// TIA Portal V20 export
FUNCTION_BLOCK "CallEquipment"   // FB44, LAD
TITLE = CallEquipment
// Template of an equipment module. This block contains the logic and futher calls (e.g. sequences, control modules, diagnostics etc.) of the equipment module.
// It can be used out of the box but also adapted to your own needs.
// stored: IsIECCheckEnabled true, MemoryReserve 100, Namespace Unit1.Em5, SetENOAutomatically true
   VAR_INPUT
      ZoneOperationEnable { ExternalWritable := 'False'} : "LWONIK_typeSafetyZoneManualOperation";
      unitEnableControlInterfaces { ExternalWritable := 'False'} : "LAF_typeEnableControlInterfaces";
      commandExcute { ExternalWritable := 'False'} : Bool;
   END_VAR
   VAR_IN_OUT
      unitStatus : "LAF_typeUnitStatus";   // Current unit status o be used in this EM
      emFeedback : "LUC_typeEmFeedback";   // Feedback of the EM to the Unit
      unitAlarmDB : "LAF_typeAlarms";   // Summarized EM Alarms for the Unit
   END_VAR
   VAR
      instSequenceManualInput { ExternalWritable := 'False'} : "Unit1.Em5.Sequence_1_ManualInput";
      instManualInPutInitializedJob1 { ExternalWritable := 'False'} : "LAF_SelectJob";
      instManualInPutLoadingJob2 { ExternalWritable := 'False'} : "LAF_SelectJob";
      instManualInPutUnLoaingJob3 { ExternalWritable := 'False'} : "LAF_SelectJob";
      instCmNgAndManualInputAxisY { ExternalWritable := 'False'} : "LBC_Axis64Pos_TecPlcCn";
      instCmMagazineAxisZ { ExternalWritable := 'False'} : "LBC_Axis64Pos_TecPlcCn";
      instCmNgAndManualInputCylinderUpDown { ExternalWritable := 'False'} : "LBC_TwoWayActuatorCn";
      instcmNgAndManualInputVacuum1OnOff { ExternalWritable := 'False'} : "LBC_TwoWayActuatorCn";
      instCmNgAndManualInputVacuum2OnOff { ExternalWritable := 'False'} : "LBC_TwoWayActuatorCn";
      instCmNgAndManualInputVibrator1OnOff { ExternalWritable := 'False'} : "LBC_TwoWayActuatorCn";
      instCmNgAndManualInputVibrator2OnOff { ExternalWritable := 'False'} : "LBC_TwoWayActuatorCn";
      instcmMagazineLockCylinderUpDown { ExternalWritable := 'False'} : "LBC_TwoWayActuatorCn";
      instCmNgAndManaulInputMagazineElectrodeDetectionSensor { ExternalWritable := 'False'} : "LBC_DigitalSignalCn";
      instCmNgAndManualInputMagazineDetectionSensor { ExternalWritable := 'False'} : "LBC_DigitalSignalCn";
      instCmNgAndManualInputMagazineFullSensor { ExternalWritable := 'False'} : "LBC_DigitalSignalCn";
      instCmNgAndManualInputElectrodeDetectionSensor { ExternalWritable := 'False'} : "LBC_DigitalSignalCn";
      instcmMagazineSafetyPinIdlePosition { ExternalWritable := 'False'} : "LBC_DigitalSignalCn";
      instNgAndManualInputAxisControlInterlockSummary { ExternalWritable := 'False'} : "LER_Axis64Pos_InterlockSummary";
      instMagazineAxisControlInterlockSummary { ExternalWritable := 'False'} : "LER_Axis64Pos_InterlockSummary";
      instServoTorqueCal_DR7 { ExternalWritable := 'False'} : "LER_ServoTorqueCal";
      instServoTorqueCal_DR8 { ExternalWritable := 'False'} : "LER_ServoTorqueCal";
      instLDrv701ControlMagazineAxisZ { ExternalWritable := 'False'} : "LDrvSafe_SinaTlg701Control";   // Drive Telegram Function Library
      instLDrv701StatusMagazineAxisZ { ExternalWritable := 'False'} : "LDrvSafe_SinaTlg701Status";   // Drive Telegram Function Library
      statUnitStatus { ExternalWritable := 'False'} : "LAF_typeUnitStatus";   // Unit Status used in this EM
      statAllBrakeTest { ExternalWritable := 'False'} : "LER_typeBrakeTestUnitCommands";
      instManageAlarms { ExternalWritable := 'False'} : "LAF_ManageAlarms";
      instEventsPFE { S7_SetPoint := 'True'} : "Unit1.Em5.EventsPFE";
      statPulse { ExternalWritable := 'False'} : Array[0..99] of Bool;
      statTonTimer { ExternalWritable := 'False'} : Array[0..99] of TON_TIME;
      statTofTimer { ExternalWritable := 'False'} : Array[0..99] of TOF_TIME;
      statEnableManualCmds { ExternalWritable := 'False'} : Bool;
      LoadingCount { ExternalWritable := 'False'} : Int;
   END_VAR
   VAR_TEMP
      tempScInProduction : Bool;   // Mode Production and StateComplete
      tempScNoProduction : Bool;   // Mode Manual and StateComplete
   END_VAR
   VAR CONSTANT
      TO_DO_INSERT_PRECONDITIONS_HERE : Bool := TRUE;   // Template : Add em specific conditions here
      NO_JOB : DInt;   // No job
      TRUE : Bool := TRUE;
      FALSE : Bool := FALSE;
      INIT_POSITION_NUMBER : SInt := -1;
      MIN_POSITION_NUMBER : SInt;
   END_VAR
   VAR_TEMP   // added for the SCL form of the ladder/FBD networks
      _w1 : Bool;
      _w2 : Bool;
      _w3 : Bool;
      _w4 : Bool;
      _w5 : Bool;
      _w6 : Bool;
      _w7 : Bool;
      _w8 : Bool;
      _w9 : Bool;
      _w10 : Bool;
      _w11 : Bool;
      _w12 : Bool;
      _w13 : Bool;
      _w14 : Bool;
      _w15 : Bool;
      _w16 : Bool;
   END_VAR
BEGIN

REGION Network 1: BLOCK INFO HEADER
   // (company) / (C) Copyright (year)
   // ---------------------------------------------------------------------------------
   // Title:                             (Title of this block)
   // Comment/Function: (that is implemented in the block)
   // Library/Family:           (that the source is dedicated to)
   // Author:                        (department / person in charge / contact)
   // Target System:          (test system with FW version)
   // Engineering:              TIA Portal (SW version)
   // Restrictions:               (OB types, etc.)
   // Requirements:           (hardware, technological package, etc.)
   // ---------------------------------------------------------------------------------
   // Change log table:
   // Version          | Date             | Signature      | Expert in charge  | Changes applied ------------------------|----------------------|-------------------------|--------------------------------|-----------------------
   // 001.000.000 | yyyy-mm-dd | 0x00000000 | (name of expert) | First released version
END_REGION

REGION Network 2: DESCRIPTION
   // This is a template block provided by the Automation Framework. It can be used to create an own project.
   // The Block Info Header is prepared to put in your own data.
   // Description of the block could be added here and the docu created by Code2Docu.
END_REGION

REGION Network 3: ******************** Unit Input ********************
END_REGION

REGION Network 4: Em Nodes Brake Test
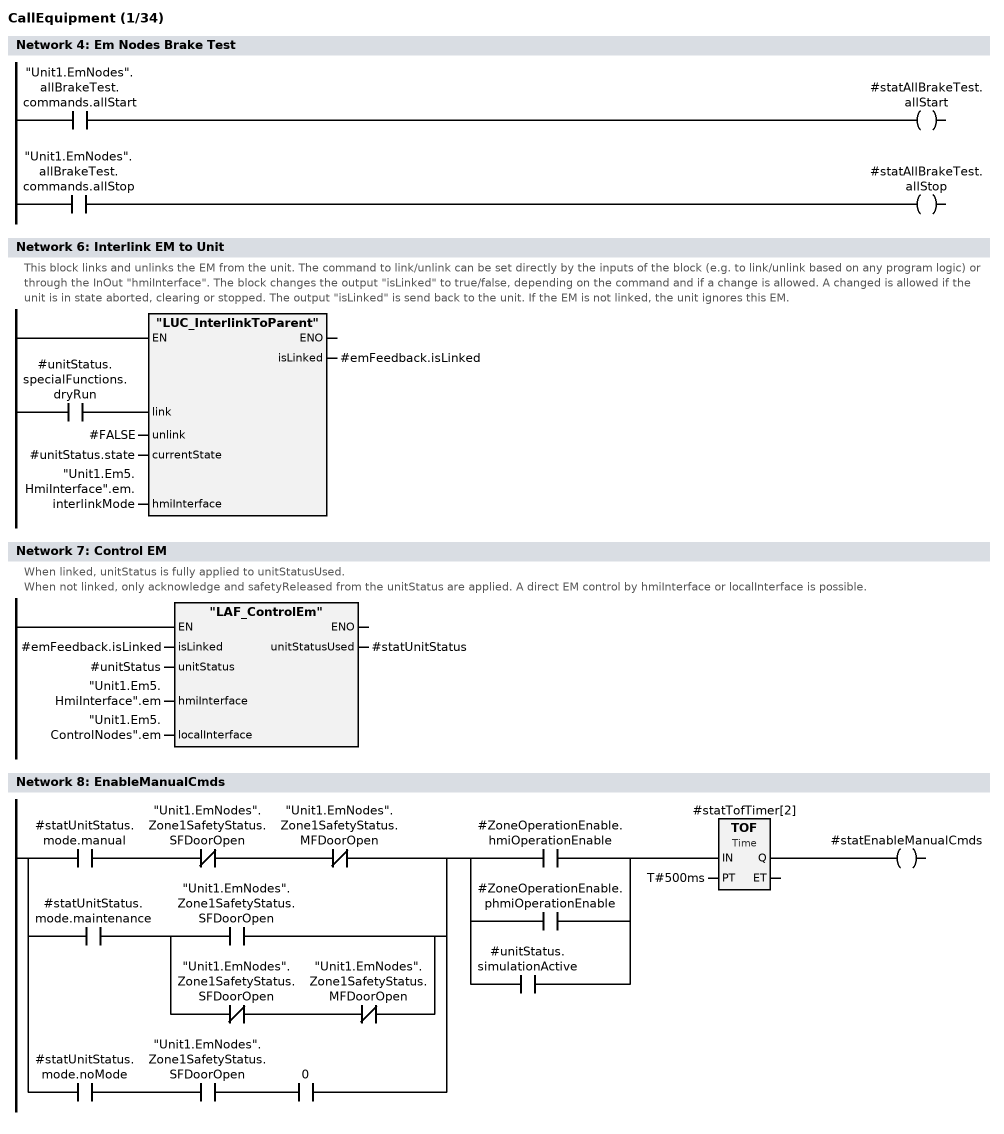
   RUNG wire#powerrail
      Contact( "Unit1.EmNodes".allBrakeTest.commands.allStart )
      Coil( #statAllBrakeTest.allStart )
   END_RUNG
   RUNG wire#powerrail
      Contact( "Unit1.EmNodes".allBrakeTest.commands.allStop )
      Coil( #statAllBrakeTest.allStop )
   END_RUNG
   // the same network as SCL:
   #statAllBrakeTest.allStart := "Unit1.EmNodes".allBrakeTest.commands.allStart;
   #statAllBrakeTest.allStop := "Unit1.EmNodes".allBrakeTest.commands.allStop;
END_REGION

REGION Network 5: ******************** Equipment Control ********************
END_REGION

REGION Network 6: Interlink EM to Unit
   // This block links and unlinks the EM from the unit. The command to link/unlink can be set directly by the inputs of the block (e.g. to link/unlink based on any program logic) or through the InOut "hmiInterface". The block changes the output "isLinked" to true/false, depending on the command and if a change is allowed. A changed is allowed if the unit is in state aborted, clearing or stopped. The output "isLinked" is send back to the unit. If the EM is not linked, the unit ignores this EM.
   RUNG wire#powerrail
      "LUC_InterlinkToParent"(link := wire#w1, unlink := #FALSE, currentState := #unitStatus.state, hmiInterface := "Unit1.Em5.HmiInterface".em.interlinkMode, isLinked => #emFeedback.isLinked)
   END_RUNG
   RUNG wire#powerrail
      Contact( #unitStatus.specialFunctions.dryRun )
   END_RUNG wire#w1
   // the same network as SCL:
   "LUC_InterlinkToParent"(link := #unitStatus.specialFunctions.dryRun,
                           unlink := #FALSE,
                           currentState := #unitStatus.state,
                           hmiInterface := "Unit1.Em5.HmiInterface".em.interlinkMode,
                           isLinked => #emFeedback.isLinked);
END_REGION

REGION Network 7: Control EM
   // When linked, unitStatus is fully applied to unitStatusUsed.
   // When not linked, only acknowledge and safetyReleased from the unitStatus are applied. A direct EM control by hmiInterface or localInterface is possible.
   RUNG wire#powerrail
      "LAF_ControlEm"(isLinked := #emFeedback.isLinked, unitStatus := #unitStatus, hmiInterface := "Unit1.Em5.HmiInterface".em, localInterface := "Unit1.Em5.ControlNodes".em, unitStatusUsed => #statUnitStatus)
   END_RUNG
   // the same network as SCL:
   "LAF_ControlEm"(isLinked := #emFeedback.isLinked,
                   unitStatus := #unitStatus,
                   hmiInterface := "Unit1.Em5.HmiInterface".em,
                   localInterface := "Unit1.Em5.ControlNodes".em,
                   unitStatusUsed => #statUnitStatus);
END_REGION

REGION Network 8: EnableManualCmds
   RUNG wire#powerrail
      Contact( #statUnitStatus.mode.manual )
      I_Contact( "Unit1.EmNodes".Zone1SafetyStatus.SFDoorOpen )
      I_Contact( "Unit1.EmNodes".Zone1SafetyStatus.MFDoorOpen )
      wire#w1
      Contact( #ZoneOperationEnable.hmiOperationEnable )
      wire#w3
      { S7_Templates := "time_type := Time" } #statTofTimer[2].TOF(pt := T#500ms, et =>)
      Coil( #statEnableManualCmds )
   END_RUNG
   RUNG wire#powerrail
      Contact( #statUnitStatus.mode.maintenance )
      wire#w2
      Contact( "Unit1.EmNodes".Zone1SafetyStatus.SFDoorOpen )
   END_RUNG wire#w1
   RUNG wire#w2
      I_Contact( "Unit1.EmNodes".Zone1SafetyStatus.SFDoorOpen )
      I_Contact( "Unit1.EmNodes".Zone1SafetyStatus.MFDoorOpen )
   END_RUNG wire#w1
   RUNG wire#powerrail
      Contact( #statUnitStatus.mode.noMode )
      Contact( "Unit1.EmNodes".Zone1SafetyStatus.SFDoorOpen )
      Contact( 0 )
   END_RUNG wire#w1
   RUNG wire#w1
      Contact( #ZoneOperationEnable.phmiOperationEnable )
   END_RUNG wire#w3
   RUNG wire#w1
      Contact( #unitStatus.simulationActive )
   END_RUNG wire#w3
   // the same network as SCL:
   #statTofTimer[2].TOF(IN := ((#statUnitStatus.mode.manual AND NOT "Unit1.EmNodes".Zone1SafetyStatus.SFDoorOpen AND NOT "Unit1.EmNodes".Zone1SafetyStatus.MFDoorOpen) OR (#statUnitStatus.mode.maintenance AND ("Unit1.EmNodes".Zone1SafetyStatus.SFDoorOpen OR (NOT "Unit1.EmNodes".Zone1SafetyStatus.SFDoorOpen AND NOT "Unit1.EmNodes".Zone1SafetyStatus.MFDoorOpen))) OR (#statUnitStatus.mode.noMode AND "Unit1.EmNodes".Zone1SafetyStatus.SFDoorOpen AND 0)) AND (#ZoneOperationEnable.hmiOperationEnable OR #ZoneOperationEnable.phmiOperationEnable OR #unitStatus.simulationActive),
                        PT := T#500ms);
   #statEnableManualCmds := #statTofTimer[2].Q;
END_REGION

REGION Network 9: Alarms Disabled
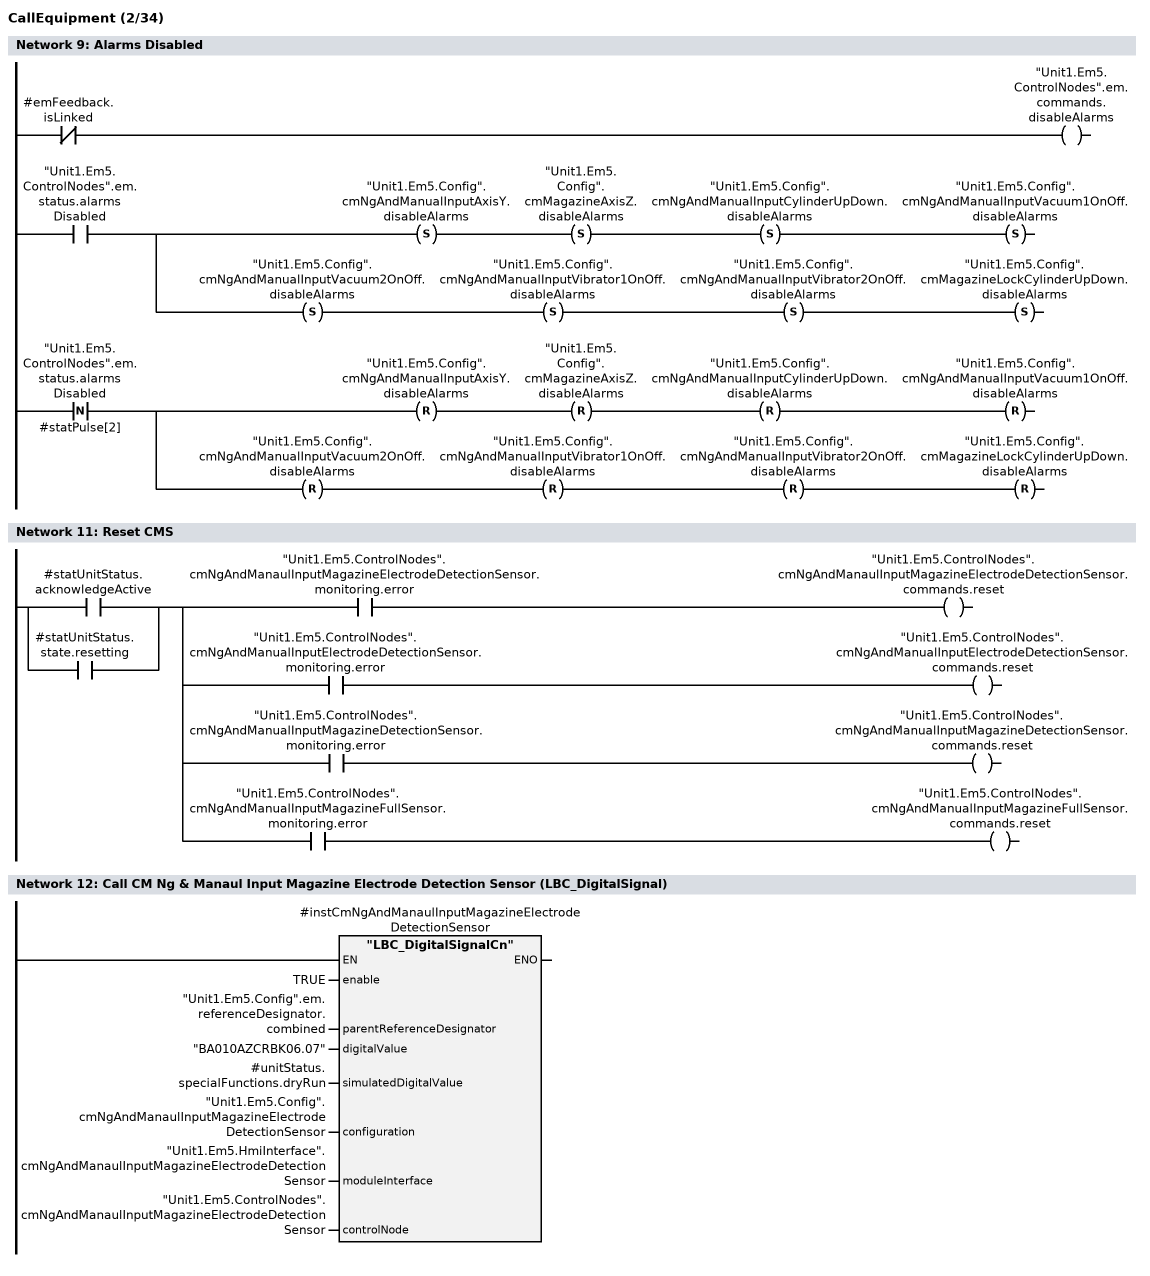
   RUNG wire#powerrail
      I_Contact( #emFeedback.isLinked )
      Coil( "Unit1.Em5.ControlNodes".em.commands.disableAlarms )
   END_RUNG
   RUNG wire#powerrail
      Contact( "Unit1.Em5.ControlNodes".em.status.alarmsDisabled )
      wire#w1
      S_Coil( "Unit1.Em5.Config".cmNgAndManualInputAxisY.disableAlarms )
      S_Coil( "Unit1.Em5.Config".cmMagazineAxisZ.disableAlarms )
      S_Coil( "Unit1.Em5.Config".cmNgAndManualInputCylinderUpDown.disableAlarms )
      S_Coil( "Unit1.Em5.Config".cmNgAndManualInputVacuum1OnOff.disableAlarms )
   END_RUNG
   RUNG wire#w1
      S_Coil( "Unit1.Em5.Config".cmNgAndManualInputVacuum2OnOff.disableAlarms )
      S_Coil( "Unit1.Em5.Config".cmNgAndManualInputVibrator1OnOff.disableAlarms )
      S_Coil( "Unit1.Em5.Config".cmNgAndManualInputVibrator2OnOff.disableAlarms )
      S_Coil( "Unit1.Em5.Config".cmMagazineLockCylinderUpDown.disableAlarms )
   END_RUNG
   RUNG wire#powerrail
      N_Contact(operand := "Unit1.Em5.ControlNodes".em.status.alarmsDisabled, bit := #statPulse[2])
      wire#w2
      R_Coil( "Unit1.Em5.Config".cmNgAndManualInputAxisY.disableAlarms )
      R_Coil( "Unit1.Em5.Config".cmMagazineAxisZ.disableAlarms )
      R_Coil( "Unit1.Em5.Config".cmNgAndManualInputCylinderUpDown.disableAlarms )
      R_Coil( "Unit1.Em5.Config".cmNgAndManualInputVacuum1OnOff.disableAlarms )
   END_RUNG
   RUNG wire#w2
      R_Coil( "Unit1.Em5.Config".cmNgAndManualInputVacuum2OnOff.disableAlarms )
      R_Coil( "Unit1.Em5.Config".cmNgAndManualInputVibrator1OnOff.disableAlarms )
      R_Coil( "Unit1.Em5.Config".cmNgAndManualInputVibrator2OnOff.disableAlarms )
      R_Coil( "Unit1.Em5.Config".cmMagazineLockCylinderUpDown.disableAlarms )
   END_RUNG
   // the same network as SCL:
   "Unit1.Em5.ControlNodes".em.commands.disableAlarms := NOT #emFeedback.isLinked;
   IF "Unit1.Em5.ControlNodes".em.status.alarmsDisabled THEN
       "Unit1.Em5.Config".cmNgAndManualInputAxisY.disableAlarms := TRUE;
       "Unit1.Em5.Config".cmMagazineAxisZ.disableAlarms := TRUE;
       "Unit1.Em5.Config".cmNgAndManualInputCylinderUpDown.disableAlarms := TRUE;
       "Unit1.Em5.Config".cmNgAndManualInputVacuum1OnOff.disableAlarms := TRUE;
       "Unit1.Em5.Config".cmNgAndManualInputVacuum2OnOff.disableAlarms := TRUE;
       "Unit1.Em5.Config".cmNgAndManualInputVibrator1OnOff.disableAlarms := TRUE;
       "Unit1.Em5.Config".cmNgAndManualInputVibrator2OnOff.disableAlarms := TRUE;
       "Unit1.Em5.Config".cmMagazineLockCylinderUpDown.disableAlarms := TRUE;
   END_IF;
   #_w1 := NOT "Unit1.Em5.ControlNodes".em.status.alarmsDisabled AND #statPulse[2];   // falling edge of "Unit1.Em5.ControlNodes".em.status.alarmsDisabled
   #statPulse[2] := "Unit1.Em5.ControlNodes".em.status.alarmsDisabled;
   IF #_w1 THEN
       "Unit1.Em5.Config".cmNgAndManualInputAxisY.disableAlarms := FALSE;
       "Unit1.Em5.Config".cmMagazineAxisZ.disableAlarms := FALSE;
       "Unit1.Em5.Config".cmNgAndManualInputCylinderUpDown.disableAlarms := FALSE;
       "Unit1.Em5.Config".cmNgAndManualInputVacuum1OnOff.disableAlarms := FALSE;
       "Unit1.Em5.Config".cmNgAndManualInputVacuum2OnOff.disableAlarms := FALSE;
       "Unit1.Em5.Config".cmNgAndManualInputVibrator1OnOff.disableAlarms := FALSE;
       "Unit1.Em5.Config".cmNgAndManualInputVibrator2OnOff.disableAlarms := FALSE;
       "Unit1.Em5.Config".cmMagazineLockCylinderUpDown.disableAlarms := FALSE;
   END_IF;
END_REGION

REGION Network 10: ******************** Control Modules (Sensors) ********************
   // Call control modules that are sensors before the em logic (jobs and sequence), so that the latest value is used in the logic.
END_REGION

REGION Network 11: Reset CMS
   RUNG wire#powerrail
      Contact( #statUnitStatus.acknowledgeActive )
      wire#w1
      Contact( "Unit1.Em5.ControlNodes".cmNgAndManaulInputMagazineElectrodeDetectionSensor.monitoring.error )
      Coil( "Unit1.Em5.ControlNodes".cmNgAndManaulInputMagazineElectrodeDetectionSensor.commands.reset )
   END_RUNG
   RUNG wire#powerrail
      Contact( #statUnitStatus.state.resetting )
   END_RUNG wire#w1
   RUNG wire#w1
      Contact( "Unit1.Em5.ControlNodes".cmNgAndManualInputElectrodeDetectionSensor.monitoring.error )
      Coil( "Unit1.Em5.ControlNodes".cmNgAndManualInputElectrodeDetectionSensor.commands.reset )
   END_RUNG
   RUNG wire#w1
      Contact( "Unit1.Em5.ControlNodes".cmNgAndManualInputMagazineDetectionSensor.monitoring.error )
      Coil( "Unit1.Em5.ControlNodes".cmNgAndManualInputMagazineDetectionSensor.commands.reset )
   END_RUNG
   RUNG wire#w1
      Contact( "Unit1.Em5.ControlNodes".cmNgAndManualInputMagazineFullSensor.monitoring.error )
      Coil( "Unit1.Em5.ControlNodes".cmNgAndManualInputMagazineFullSensor.commands.reset )
   END_RUNG
   // the same network as SCL:
   #_w1 := #statUnitStatus.acknowledgeActive OR #statUnitStatus.state.resetting;
   "Unit1.Em5.ControlNodes".cmNgAndManaulInputMagazineElectrodeDetectionSensor.commands.reset := #_w1 AND "Unit1.Em5.ControlNodes".cmNgAndManaulInputMagazineElectrodeDetectionSensor.monitoring.error;
   "Unit1.Em5.ControlNodes".cmNgAndManualInputElectrodeDetectionSensor.commands.reset := #_w1 AND "Unit1.Em5.ControlNodes".cmNgAndManualInputElectrodeDetectionSensor.monitoring.error;
   "Unit1.Em5.ControlNodes".cmNgAndManualInputMagazineDetectionSensor.commands.reset := #_w1 AND "Unit1.Em5.ControlNodes".cmNgAndManualInputMagazineDetectionSensor.monitoring.error;
   "Unit1.Em5.ControlNodes".cmNgAndManualInputMagazineFullSensor.commands.reset := #_w1 AND "Unit1.Em5.ControlNodes".cmNgAndManualInputMagazineFullSensor.monitoring.error;
END_REGION

REGION Network 12: Call CM Ng & Manaul Input Magazine Electrode Detection Sensor (LBC_DigitalSignal)
   RUNG wire#powerrail
      #instCmNgAndManaulInputMagazineElectrodeDetectionSensor(enable := TRUE, parentReferenceDesignator := "Unit1.Em5.Config".em.referenceDesignator.combined, digitalValue := "BA010AZCRBK06.07", simulatedDigitalValue := #unitStatus.specialFunctions.dryRun, configuration := "Unit1.Em5.Config".cmNgAndManaulInputMagazineElectrodeDetectionSensor, moduleInterface := "Unit1.Em5.HmiInterface".cmNgAndManaulInputMagazineElectrodeDetectionSensor, controlNode := "Unit1.Em5.ControlNodes".cmNgAndManaulInputMagazineElectrodeDetectionSensor)
   END_RUNG
   // the same network as SCL:
   #instCmNgAndManaulInputMagazineElectrodeDetectionSensor(enable := TRUE,   // "LBC_DigitalSignalCn"
                           parentReferenceDesignator := "Unit1.Em5.Config".em.referenceDesignator.combined,
                           digitalValue := "BA010AZCRBK06.07",
                           simulatedDigitalValue := #unitStatus.specialFunctions.dryRun,
                           configuration := "Unit1.Em5.Config".cmNgAndManaulInputMagazineElectrodeDetectionSensor,
                           moduleInterface := "Unit1.Em5.HmiInterface".cmNgAndManaulInputMagazineElectrodeDetectionSensor,
                           controlNode := "Unit1.Em5.ControlNodes".cmNgAndManaulInputMagazineElectrodeDetectionSensor);
END_REGION

REGION Network 13: Call CM Ng & Manaul Input Magazine Detection Sensor (LBC_DigitalSignal)
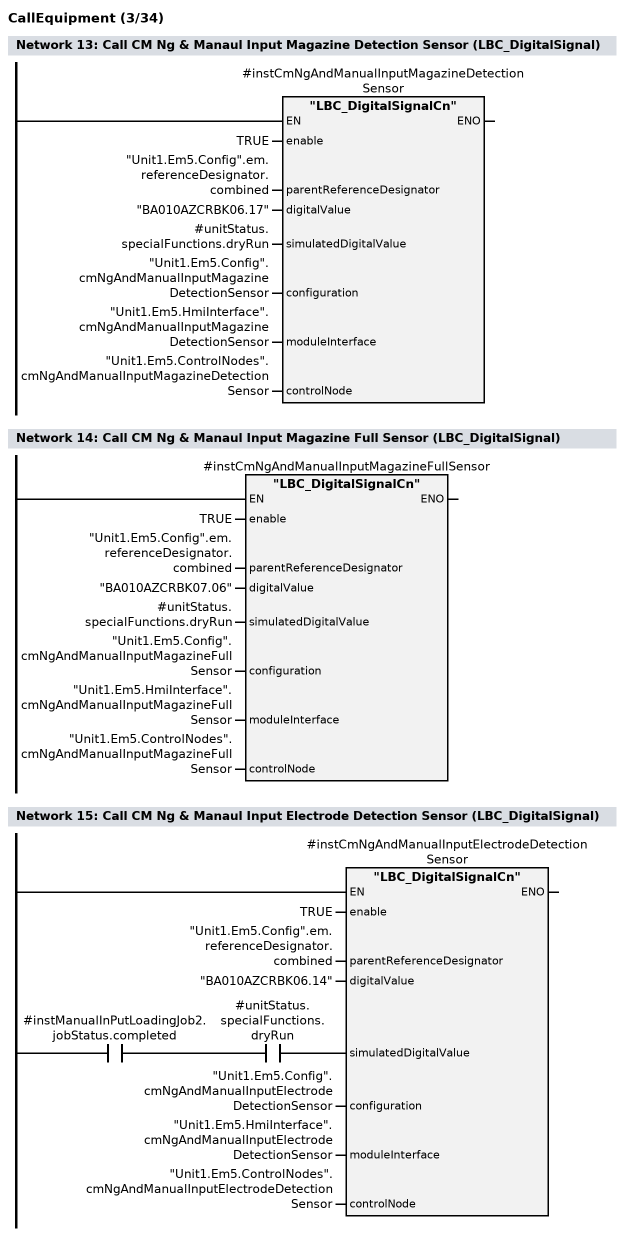
   RUNG wire#powerrail
      #instCmNgAndManualInputMagazineDetectionSensor(enable := TRUE, parentReferenceDesignator := "Unit1.Em5.Config".em.referenceDesignator.combined, digitalValue := "BA010AZCRBK06.17", simulatedDigitalValue := #unitStatus.specialFunctions.dryRun, configuration := "Unit1.Em5.Config".cmNgAndManualInputMagazineDetectionSensor, moduleInterface := "Unit1.Em5.HmiInterface".cmNgAndManualInputMagazineDetectionSensor, controlNode := "Unit1.Em5.ControlNodes".cmNgAndManualInputMagazineDetectionSensor)
   END_RUNG
   // the same network as SCL:
   #instCmNgAndManualInputMagazineDetectionSensor(enable := TRUE,   // "LBC_DigitalSignalCn"
                           parentReferenceDesignator := "Unit1.Em5.Config".em.referenceDesignator.combined,
                           digitalValue := "BA010AZCRBK06.17",
                           simulatedDigitalValue := #unitStatus.specialFunctions.dryRun,
                           configuration := "Unit1.Em5.Config".cmNgAndManualInputMagazineDetectionSensor,
                           moduleInterface := "Unit1.Em5.HmiInterface".cmNgAndManualInputMagazineDetectionSensor,
                           controlNode := "Unit1.Em5.ControlNodes".cmNgAndManualInputMagazineDetectionSensor);
END_REGION

REGION Network 14: Call CM Ng & Manaul Input Magazine Full Sensor (LBC_DigitalSignal)
   RUNG wire#powerrail
      #instCmNgAndManualInputMagazineFullSensor(enable := TRUE, parentReferenceDesignator := "Unit1.Em5.Config".em.referenceDesignator.combined, digitalValue := "BA010AZCRBK07.06", simulatedDigitalValue := #unitStatus.specialFunctions.dryRun, configuration := "Unit1.Em5.Config".cmNgAndManualInputMagazineFullSensor, moduleInterface := "Unit1.Em5.HmiInterface".cmNgAndManualInputMagazineFullSensor, controlNode := "Unit1.Em5.ControlNodes".cmNgAndManualInputMagazineFullSensor)
   END_RUNG
   // the same network as SCL:
   #instCmNgAndManualInputMagazineFullSensor(enable := TRUE,   // "LBC_DigitalSignalCn"
                           parentReferenceDesignator := "Unit1.Em5.Config".em.referenceDesignator.combined,
                           digitalValue := "BA010AZCRBK07.06",
                           simulatedDigitalValue := #unitStatus.specialFunctions.dryRun,
                           configuration := "Unit1.Em5.Config".cmNgAndManualInputMagazineFullSensor,
                           moduleInterface := "Unit1.Em5.HmiInterface".cmNgAndManualInputMagazineFullSensor,
                           controlNode := "Unit1.Em5.ControlNodes".cmNgAndManualInputMagazineFullSensor);
END_REGION

REGION Network 15: Call CM Ng & Manaul Input Electrode Detection Sensor (LBC_DigitalSignal)
   RUNG wire#powerrail
      #instCmNgAndManualInputElectrodeDetectionSensor(simulatedDigitalValue := wire#w1, enable := TRUE, parentReferenceDesignator := "Unit1.Em5.Config".em.referenceDesignator.combined, digitalValue := "BA010AZCRBK06.14", configuration := "Unit1.Em5.Config".cmNgAndManualInputElectrodeDetectionSensor, moduleInterface := "Unit1.Em5.HmiInterface".cmNgAndManualInputElectrodeDetectionSensor, controlNode := "Unit1.Em5.ControlNodes".cmNgAndManualInputElectrodeDetectionSensor)
   END_RUNG
   RUNG wire#powerrail
      Contact( #instManualInPutLoadingJob2.jobStatus.completed )
      Contact( #unitStatus.specialFunctions.dryRun )
   END_RUNG wire#w1
   // the same network as SCL:
   #instCmNgAndManualInputElectrodeDetectionSensor(enable := TRUE,   // "LBC_DigitalSignalCn"
                           parentReferenceDesignator := "Unit1.Em5.Config".em.referenceDesignator.combined,
                           digitalValue := "BA010AZCRBK06.14",
                           simulatedDigitalValue := #instManualInPutLoadingJob2.jobStatus.completed AND #unitStatus.specialFunctions.dryRun,
                           configuration := "Unit1.Em5.Config".cmNgAndManualInputElectrodeDetectionSensor,
                           moduleInterface := "Unit1.Em5.HmiInterface".cmNgAndManualInputElectrodeDetectionSensor,
                           controlNode := "Unit1.Em5.ControlNodes".cmNgAndManualInputElectrodeDetectionSensor);
END_REGION

REGION Network 16: Call CM Magazine Safety Pin Idle Position (LBC_DigitalSignal)
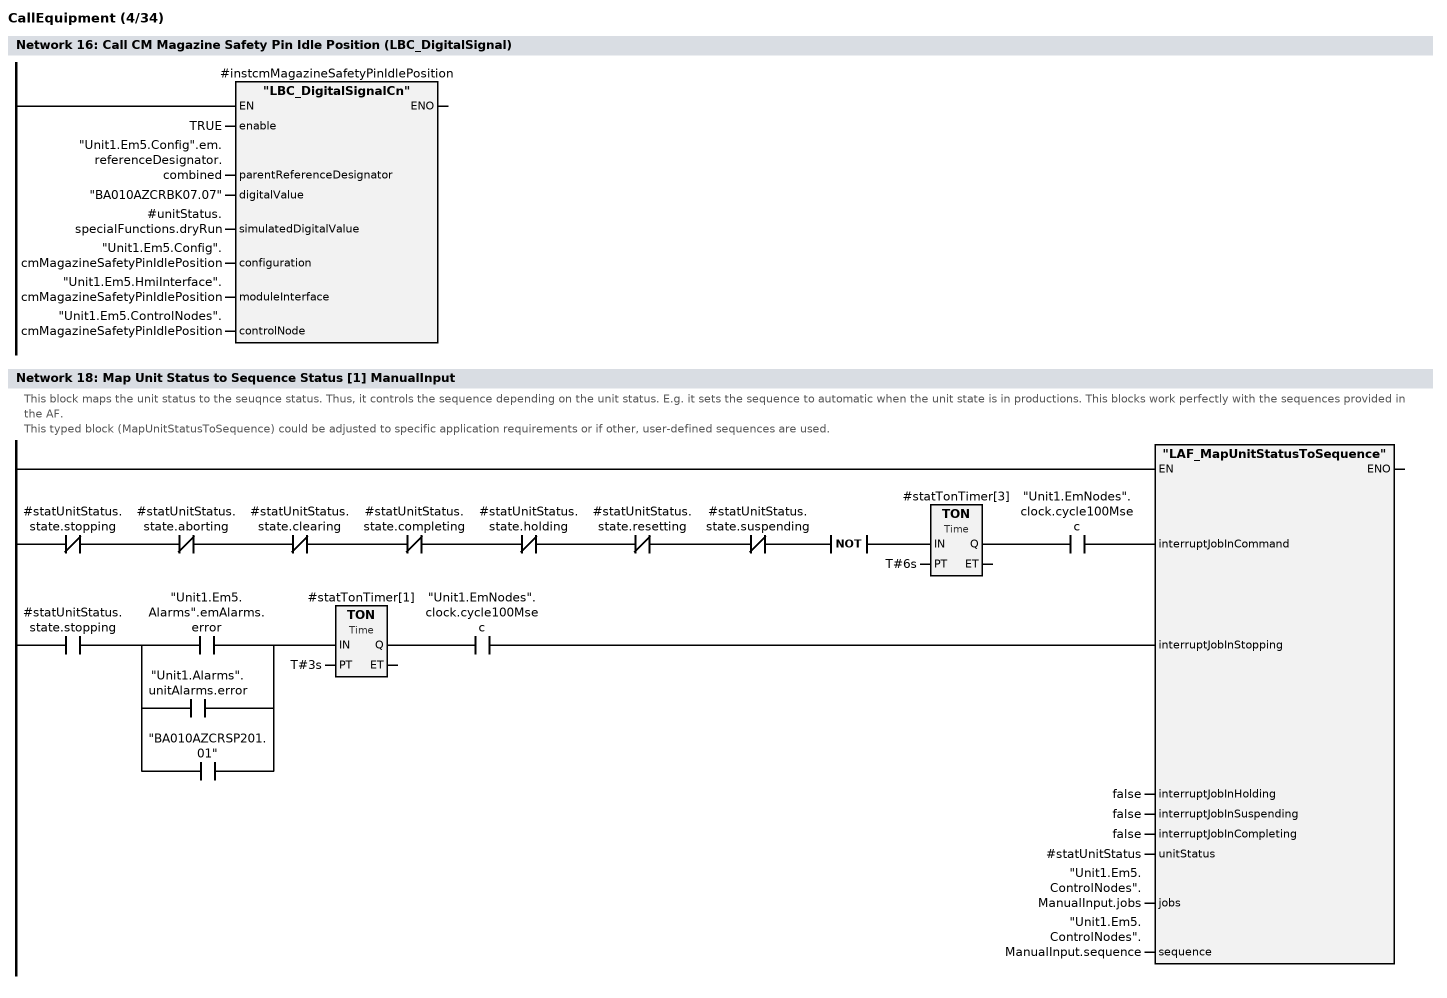
   RUNG wire#powerrail
      #instcmMagazineSafetyPinIdlePosition(enable := TRUE, parentReferenceDesignator := "Unit1.Em5.Config".em.referenceDesignator.combined, digitalValue := "BA010AZCRBK07.07", simulatedDigitalValue := #unitStatus.specialFunctions.dryRun, configuration := "Unit1.Em5.Config".cmMagazineSafetyPinIdlePosition, moduleInterface := "Unit1.Em5.HmiInterface".cmMagazineSafetyPinIdlePosition, controlNode := "Unit1.Em5.ControlNodes".cmMagazineSafetyPinIdlePosition)
   END_RUNG
   // the same network as SCL:
   #instcmMagazineSafetyPinIdlePosition(enable := TRUE,   // "LBC_DigitalSignalCn"
                           parentReferenceDesignator := "Unit1.Em5.Config".em.referenceDesignator.combined,
                           digitalValue := "BA010AZCRBK07.07",
                           simulatedDigitalValue := #unitStatus.specialFunctions.dryRun,
                           configuration := "Unit1.Em5.Config".cmMagazineSafetyPinIdlePosition,
                           moduleInterface := "Unit1.Em5.HmiInterface".cmMagazineSafetyPinIdlePosition,
                           controlNode := "Unit1.Em5.ControlNodes".cmMagazineSafetyPinIdlePosition);
END_REGION

REGION Network 17: ******************** Equipment Logic ********************
END_REGION

REGION Network 18: Map Unit Status to Sequence Status [1] ManualInput
   // This block maps the unit status to the seuqnce status. Thus, it controls the sequence depending on the unit status. E.g. it sets the sequence to automatic when the unit state is in productions. This blocks work perfectly with the sequences provided in the AF. 
   // This typed block (MapUnitStatusToSequence) could be adjusted to specific application requirements or if other, user-defined sequences are used.
   RUNG wire#powerrail
      "LAF_MapUnitStatusToSequence"(interruptJobInCommand := wire#w1, interruptJobInStopping := wire#w4, interruptJobInHolding := false, interruptJobInSuspending := false, interruptJobInCompleting := false, unitStatus := #statUnitStatus, jobs := "Unit1.Em5.ControlNodes".ManualInput.jobs, sequence := "Unit1.Em5.ControlNodes".ManualInput.sequence)
   END_RUNG
   RUNG wire#powerrail
      I_Contact( #statUnitStatus.state.stopping )
      I_Contact( #statUnitStatus.state.aborting )
      I_Contact( #statUnitStatus.state.clearing )
      I_Contact( #statUnitStatus.state.completing )
      I_Contact( #statUnitStatus.state.holding )
      I_Contact( #statUnitStatus.state.resetting )
      I_Contact( #statUnitStatus.state.suspending )
      Not()
      { S7_Templates := "time_type := Time" } #statTonTimer[3].TON(pt := T#6s, et =>)
      Contact( "Unit1.EmNodes".clock.cycle100Msec )
   END_RUNG wire#w1
   RUNG wire#powerrail
      Contact( #statUnitStatus.state.stopping )
      wire#w2
      Contact( "Unit1.Em5.Alarms".emAlarms.error )
      wire#w3
      { S7_Templates := "time_type := Time" } #statTonTimer[1].TON(pt := T#3s, et =>)
      Contact( "Unit1.EmNodes".clock.cycle100Msec )
   END_RUNG wire#w4
   RUNG wire#w2
      Contact( "Unit1.Alarms".unitAlarms.error )
   END_RUNG wire#w3
   RUNG wire#w2
      Contact( "BA010AZCRSP201.01" )
   END_RUNG wire#w3
   // the same network as SCL:
   #statTonTimer[3].TON(IN := NOT (NOT #statUnitStatus.state.stopping AND NOT #statUnitStatus.state.aborting AND NOT #statUnitStatus.state.clearing AND NOT #statUnitStatus.state.completing AND NOT #statUnitStatus.state.holding AND NOT #statUnitStatus.state.resetting AND NOT #statUnitStatus.state.suspending),
                        PT := T#6s);
   #_w1 := #statTonTimer[3].Q AND "Unit1.EmNodes".clock.cycle100Msec;
   #statTonTimer[1].TON(IN := #statUnitStatus.state.stopping AND ("Unit1.Em5.Alarms".emAlarms.error OR "Unit1.Alarms".unitAlarms.error OR "BA010AZCRSP201.01"),
                        PT := T#3s);
   "LAF_MapUnitStatusToSequence"(interruptJobInCommand := #_w1,
                           interruptJobInStopping := #statTonTimer[1].Q AND "Unit1.EmNodes".clock.cycle100Msec,
                           interruptJobInHolding := false,
                           interruptJobInSuspending := false,
                           interruptJobInCompleting := false,
                           unitStatus := #statUnitStatus,
                           jobs := "Unit1.Em5.ControlNodes".ManualInput.jobs,
                           sequence := "Unit1.Em5.ControlNodes".ManualInput.sequence);
END_REGION

REGION Network 19: Select Job [1] ManualInput Initialized
   // Decide which Step Sequence to start depending on the OMAC State and EM conditions
   // First Move Block is to Initialize the jobSelect Number
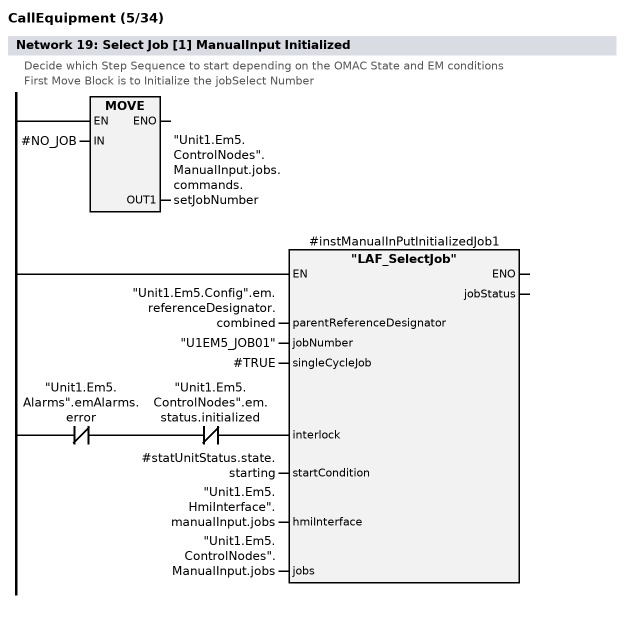
   RUNG wire#powerrail
      Move(in := #NO_JOB, out1 => "Unit1.Em5.ControlNodes".ManualInput.jobs.commands.setJobNumber)
   END_RUNG
   RUNG wire#powerrail
      #instManualInPutInitializedJob1(interlock := wire#w1, parentReferenceDesignator := "Unit1.Em5.Config".em.referenceDesignator.combined, jobNumber := "U1EM5_JOB01", singleCycleJob := #TRUE, startCondition := #statUnitStatus.state.starting, hmiInterface := "Unit1.Em5.HmiInterface".manualInput.jobs, jobs := "Unit1.Em5.ControlNodes".ManualInput.jobs, jobStatus =>)
   END_RUNG
   RUNG wire#powerrail
      I_Contact( "Unit1.Em5.Alarms".emAlarms.error )
      I_Contact( "Unit1.Em5.ControlNodes".em.status.initialized )
   END_RUNG wire#w1
   // the same network as SCL:
   "Unit1.Em5.ControlNodes".ManualInput.jobs.commands.setJobNumber := #NO_JOB;
   #instManualInPutInitializedJob1(parentReferenceDesignator := "Unit1.Em5.Config".em.referenceDesignator.combined,   // "LAF_SelectJob"
                           jobNumber := "U1EM5_JOB01",
                           singleCycleJob := #TRUE,
                           interlock := NOT "Unit1.Em5.Alarms".emAlarms.error AND NOT "Unit1.Em5.ControlNodes".em.status.initialized,
                           startCondition := #statUnitStatus.state.starting,
                           hmiInterface := "Unit1.Em5.HmiInterface".manualInput.jobs,
                           jobs := "Unit1.Em5.ControlNodes".ManualInput.jobs);
END_REGION

REGION Network 20: Select Job [2] Loading Auto
   // Decide which Step Sequence to start depending on the OMAC State and EM conditions
   // First Move Block is to Initialize the jobSelect Number
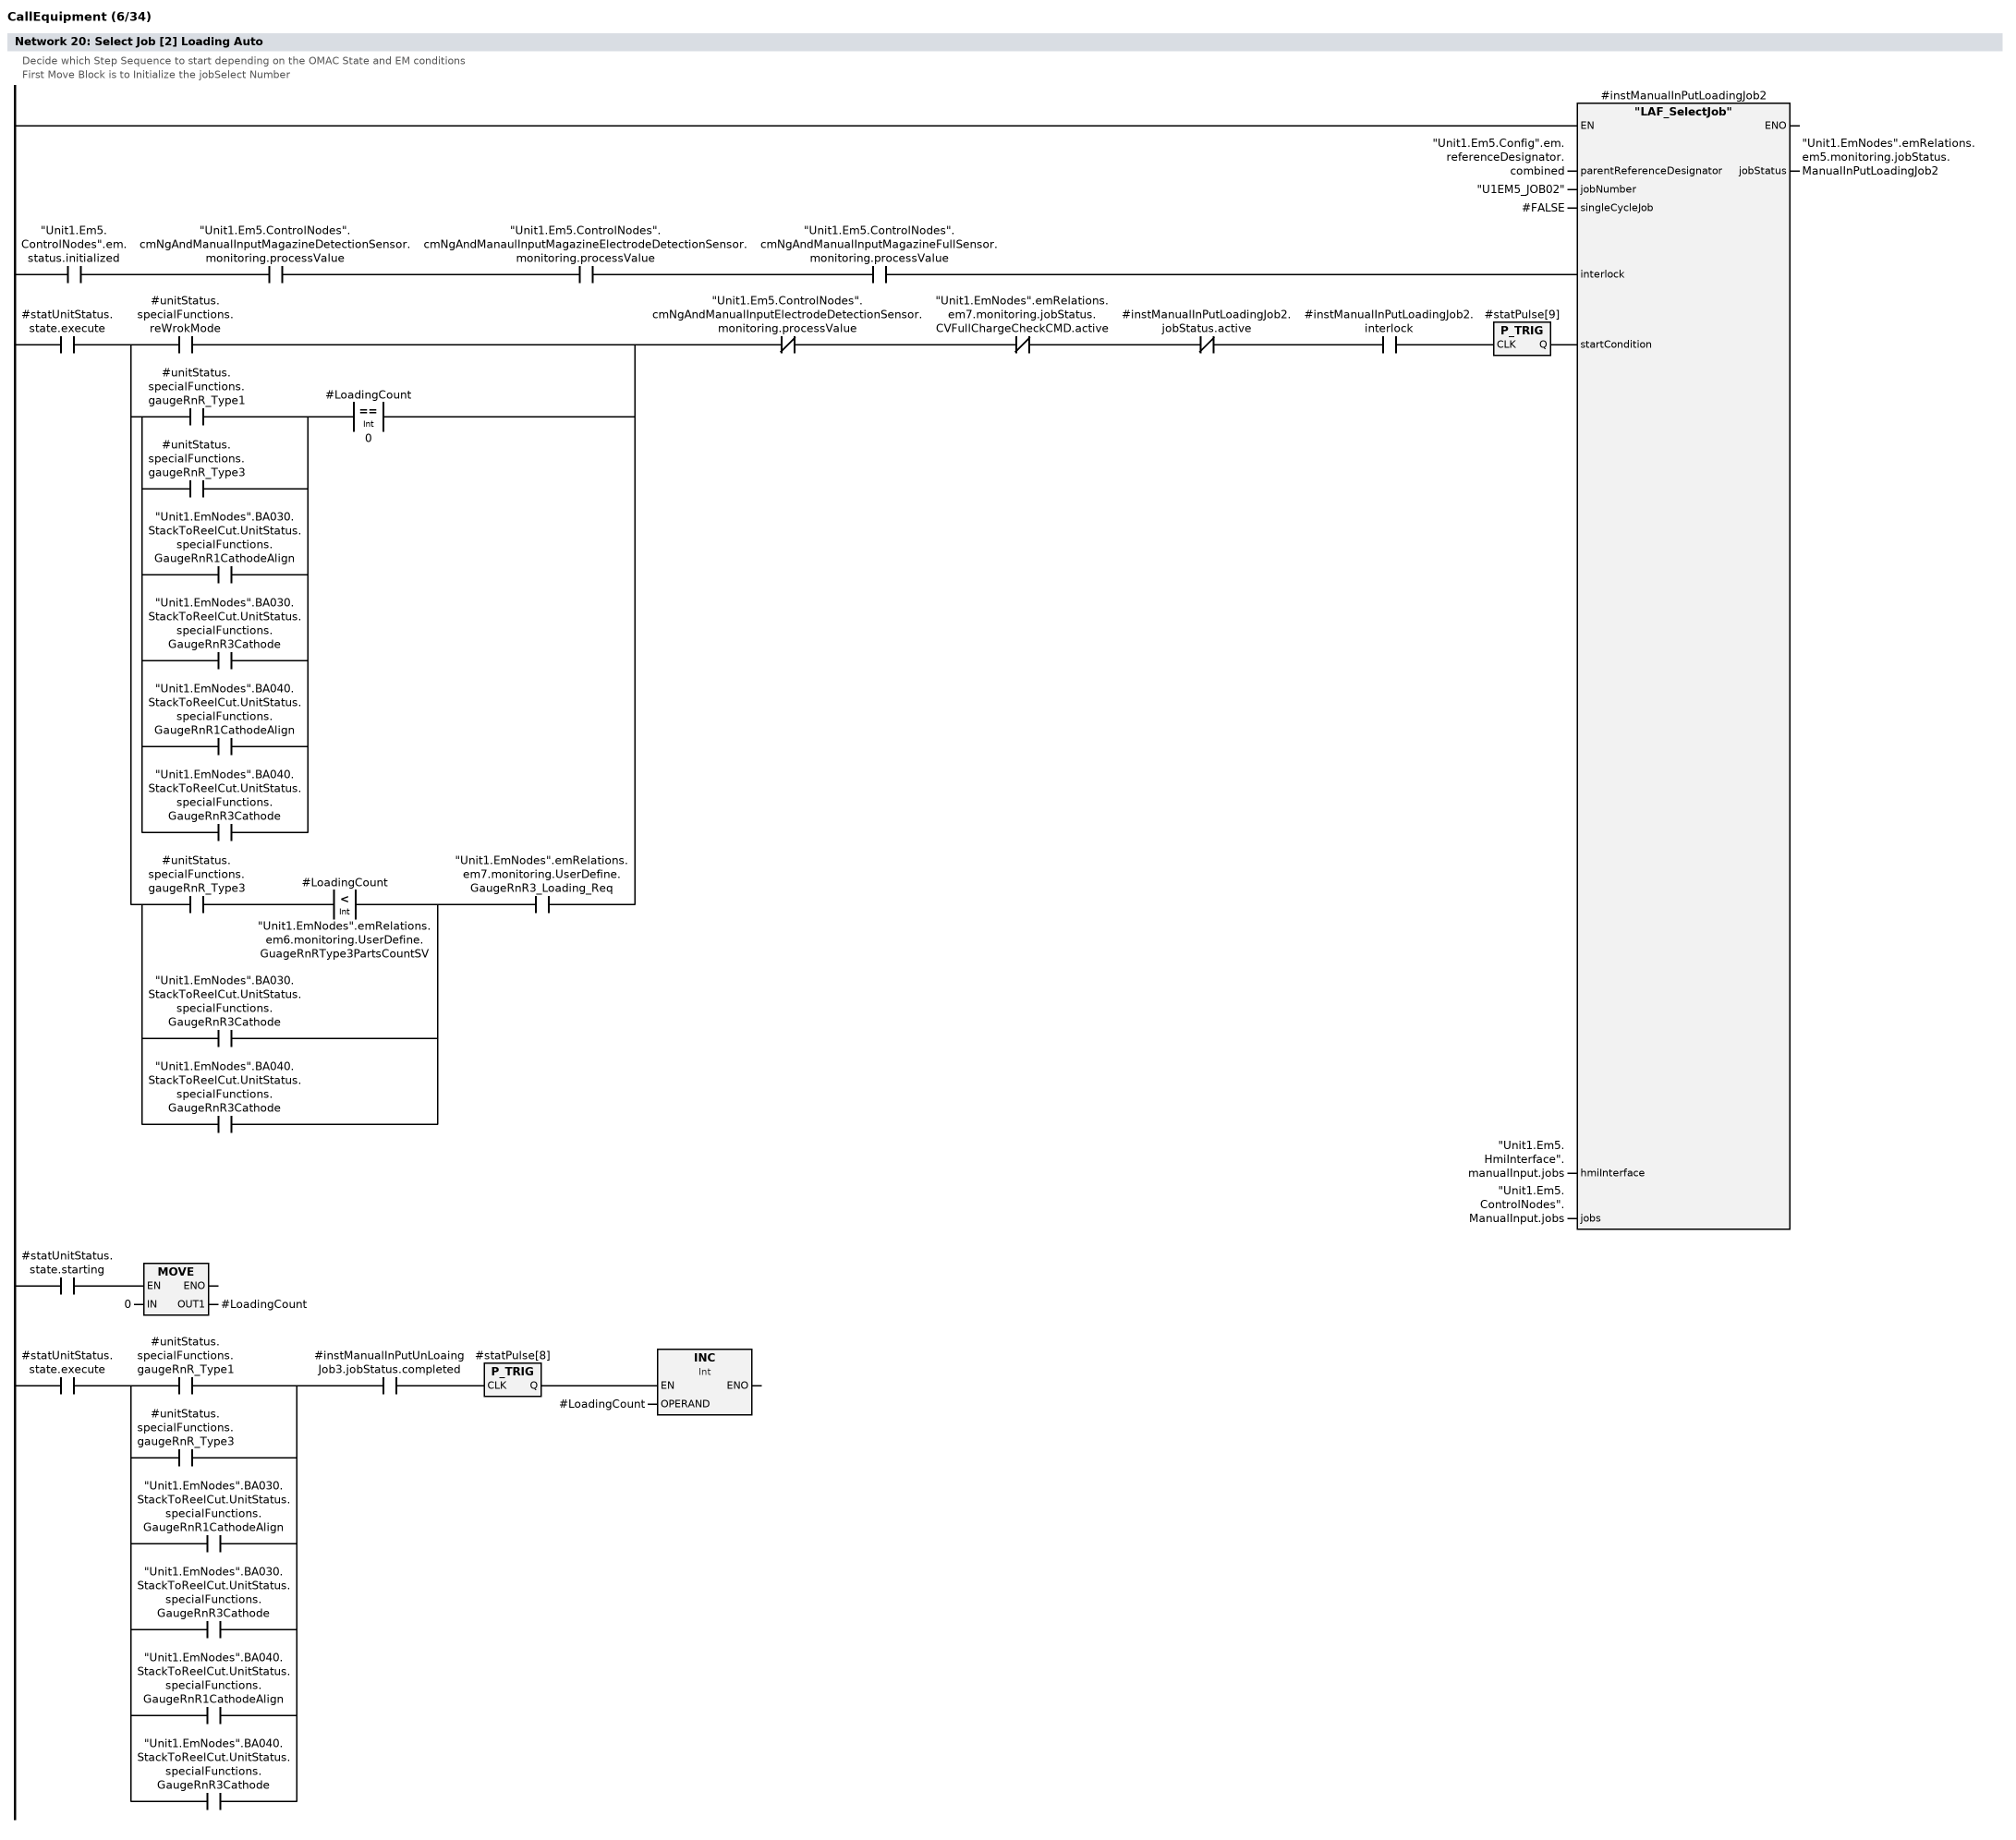
   RUNG wire#powerrail
      #instManualInPutLoadingJob2(interlock := wire#w1, startCondition := wire#w6, parentReferenceDesignator := "Unit1.Em5.Config".em.referenceDesignator.combined, jobNumber := "U1EM5_JOB02", singleCycleJob := #FALSE, hmiInterface := "Unit1.Em5.HmiInterface".manualInput.jobs, jobs := "Unit1.Em5.ControlNodes".ManualInput.jobs, jobStatus => "Unit1.EmNodes".emRelations.em5.monitoring.jobStatus.ManualInPutLoadingJob2)
   END_RUNG
   RUNG wire#powerrail
      Contact( "Unit1.Em5.ControlNodes".em.status.initialized )
      Contact( "Unit1.Em5.ControlNodes".cmNgAndManualInputMagazineDetectionSensor.monitoring.processValue )
      Contact( "Unit1.Em5.ControlNodes".cmNgAndManaulInputMagazineElectrodeDetectionSensor.monitoring.processValue )
      Contact( "Unit1.Em5.ControlNodes".cmNgAndManualInputMagazineFullSensor.monitoring.processValue )
   END_RUNG wire#w1
   RUNG wire#powerrail
      Contact( #statUnitStatus.state.execute )
      wire#w2
      Contact( #unitStatus.specialFunctions.reWrokMode )
      wire#w3
      I_Contact( "Unit1.Em5.ControlNodes".cmNgAndManualInputElectrodeDetectionSensor.monitoring.processValue )
      I_Contact( "Unit1.EmNodes".emRelations.em7.monitoring.jobStatus.CVFullChargeCheckCMD.active )
      I_Contact( #instManualInPutLoadingJob2.jobStatus.active )
      Contact( #instManualInPutLoadingJob2.interlock )
      P_Trig( #statPulse[9] )
   END_RUNG wire#w6
   RUNG wire#w2
      Contact( #unitStatus.specialFunctions.gaugeRnR_Type1 )
      wire#w4
      { S7_Templates := "SrcType := Int" } EQ_Contact(in1 := #LoadingCount, in2 := 0)
   END_RUNG wire#w3
   RUNG wire#w2
      Contact( #unitStatus.specialFunctions.gaugeRnR_Type3 )
   END_RUNG wire#w4
   RUNG wire#w2
      Contact( "Unit1.EmNodes".BA030.StackToReelCut.UnitStatus.specialFunctions.GaugeRnR1CathodeAlign )
   END_RUNG wire#w4
   RUNG wire#w2
      Contact( "Unit1.EmNodes".BA030.StackToReelCut.UnitStatus.specialFunctions.GaugeRnR3Cathode )
   END_RUNG wire#w4
   RUNG wire#w2
      Contact( "Unit1.EmNodes".BA040.StackToReelCut.UnitStatus.specialFunctions.GaugeRnR1CathodeAlign )
   END_RUNG wire#w4
   RUNG wire#w2
      Contact( "Unit1.EmNodes".BA040.StackToReelCut.UnitStatus.specialFunctions.GaugeRnR3Cathode )
   END_RUNG wire#w4
   RUNG wire#w2
      Contact( #unitStatus.specialFunctions.gaugeRnR_Type3 )
      { S7_Templates := "SrcType := Int" } LT_Contact(in1 := #LoadingCount, in2 := "Unit1.EmNodes".emRelations.em6.monitoring.UserDefine.GuageRnRType3PartsCountSV)
      wire#w5
      Contact( "Unit1.EmNodes".emRelations.em7.monitoring.UserDefine.GaugeRnR3_Loading_Req )
   END_RUNG wire#w3
   RUNG wire#w2
      Contact( "Unit1.EmNodes".BA030.StackToReelCut.UnitStatus.specialFunctions.GaugeRnR3Cathode )
   END_RUNG wire#w5
   RUNG wire#w2
      Contact( "Unit1.EmNodes".BA040.StackToReelCut.UnitStatus.specialFunctions.GaugeRnR3Cathode )
   END_RUNG wire#w5
   RUNG wire#powerrail
      Contact( #statUnitStatus.state.starting )
      Move(in := 0, out1 => #LoadingCount)
   END_RUNG
   RUNG wire#powerrail
      Contact( #statUnitStatus.state.execute )
      wire#w7
      Contact( #unitStatus.specialFunctions.gaugeRnR_Type1 )
      wire#w8
      Contact( #instManualInPutUnLoaingJob3.jobStatus.completed )
      P_Trig( #statPulse[8] )
      { S7_Templates := "DestType := Int" } Inc( #LoadingCount )
   END_RUNG
   RUNG wire#w7
      Contact( #unitStatus.specialFunctions.gaugeRnR_Type3 )
   END_RUNG wire#w8
   RUNG wire#w7
      Contact( "Unit1.EmNodes".BA030.StackToReelCut.UnitStatus.specialFunctions.GaugeRnR1CathodeAlign )
   END_RUNG wire#w8
   RUNG wire#w7
      Contact( "Unit1.EmNodes".BA030.StackToReelCut.UnitStatus.specialFunctions.GaugeRnR3Cathode )
   END_RUNG wire#w8
   RUNG wire#w7
      Contact( "Unit1.EmNodes".BA040.StackToReelCut.UnitStatus.specialFunctions.GaugeRnR1CathodeAlign )
   END_RUNG wire#w8
   RUNG wire#w7
      Contact( "Unit1.EmNodes".BA040.StackToReelCut.UnitStatus.specialFunctions.GaugeRnR3Cathode )
   END_RUNG wire#w8
   // the same network as SCL:
   #_w1 := #statUnitStatus.state.execute AND (#unitStatus.specialFunctions.reWrokMode OR ((#unitStatus.specialFunctions.gaugeRnR_Type1 OR #unitStatus.specialFunctions.gaugeRnR_Type3 OR "Unit1.EmNodes".BA030.StackToReelCut.UnitStatus.specialFunctions.GaugeRnR1CathodeAlign OR "Unit1.EmNodes".BA030.StackToReelCut.UnitStatus.specialFunctions.GaugeRnR3Cathode OR "Unit1.EmNodes".BA040.StackToReelCut.UnitStatus.specialFunctions.GaugeRnR1CathodeAlign OR "Unit1.EmNodes".BA040.StackToReelCut.UnitStatus.specialFunctions.GaugeRnR3Cathode) AND (#LoadingCount = 0)) OR (((#unitStatus.specialFunctions.gaugeRnR_Type3 AND (#LoadingCount < "Unit1.EmNodes".emRelations.em6.monitoring.UserDefine.GuageRnRType3PartsCountSV)) OR "Unit1.EmNodes".BA030.StackToReelCut.UnitStatus.specialFunctions.GaugeRnR3Cathode OR "Unit1.EmNodes".BA040.StackToReelCut.UnitStatus.specialFunctions.GaugeRnR3Cathode) AND "Unit1.EmNodes".emRelations.em7.monitoring.UserDefine.GaugeRnR3_Loading_Req)) AND NOT "Unit1.Em5.ControlNodes".cmNgAndManualInputElectrodeDetectionSensor.monitoring.processValue AND NOT "Unit1.EmNodes".emRelations.em7.monitoring.jobStatus.CVFullChargeCheckCMD.active AND NOT #instManualInPutLoadingJob2.jobStatus.active AND #instManualInPutLoadingJob2.interlock;
   #_w2 := #_w1 AND NOT #statPulse[9];   // rising edge
   #statPulse[9] := #_w1;
   #instManualInPutLoadingJob2(parentReferenceDesignator := "Unit1.Em5.Config".em.referenceDesignator.combined,   // "LAF_SelectJob"
                           jobNumber := "U1EM5_JOB02",
                           singleCycleJob := #FALSE,
                           interlock := "Unit1.Em5.ControlNodes".em.status.initialized AND "Unit1.Em5.ControlNodes".cmNgAndManualInputMagazineDetectionSensor.monitoring.processValue AND "Unit1.Em5.ControlNodes".cmNgAndManaulInputMagazineElectrodeDetectionSensor.monitoring.processValue AND "Unit1.Em5.ControlNodes".cmNgAndManualInputMagazineFullSensor.monitoring.processValue,
                           startCondition := #_w2,
                           hmiInterface := "Unit1.Em5.HmiInterface".manualInput.jobs,
                           jobs := "Unit1.Em5.ControlNodes".ManualInput.jobs,
                           jobStatus => "Unit1.EmNodes".emRelations.em5.monitoring.jobStatus.ManualInPutLoadingJob2);
   IF #statUnitStatus.state.starting THEN #LoadingCount := 0; END_IF;
   #_w3 := #statUnitStatus.state.execute AND (#unitStatus.specialFunctions.gaugeRnR_Type1 OR #unitStatus.specialFunctions.gaugeRnR_Type3 OR "Unit1.EmNodes".BA030.StackToReelCut.UnitStatus.specialFunctions.GaugeRnR1CathodeAlign OR "Unit1.EmNodes".BA030.StackToReelCut.UnitStatus.specialFunctions.GaugeRnR3Cathode OR "Unit1.EmNodes".BA040.StackToReelCut.UnitStatus.specialFunctions.GaugeRnR1CathodeAlign OR "Unit1.EmNodes".BA040.StackToReelCut.UnitStatus.specialFunctions.GaugeRnR3Cathode) AND #instManualInPutUnLoaingJob3.jobStatus.completed;
   #_w4 := #_w3 AND NOT #statPulse[8];   // rising edge
   #statPulse[8] := #_w3;
   IF #_w4 THEN #LoadingCount := #LoadingCount + 1; END_IF;
END_REGION

REGION Network 21: Select Job [3] UnLoading Auto
   // Decide which Step Sequence to start depending on the OMAC State and EM conditions
   // First Move Block is to Initialize the jobSelect Number
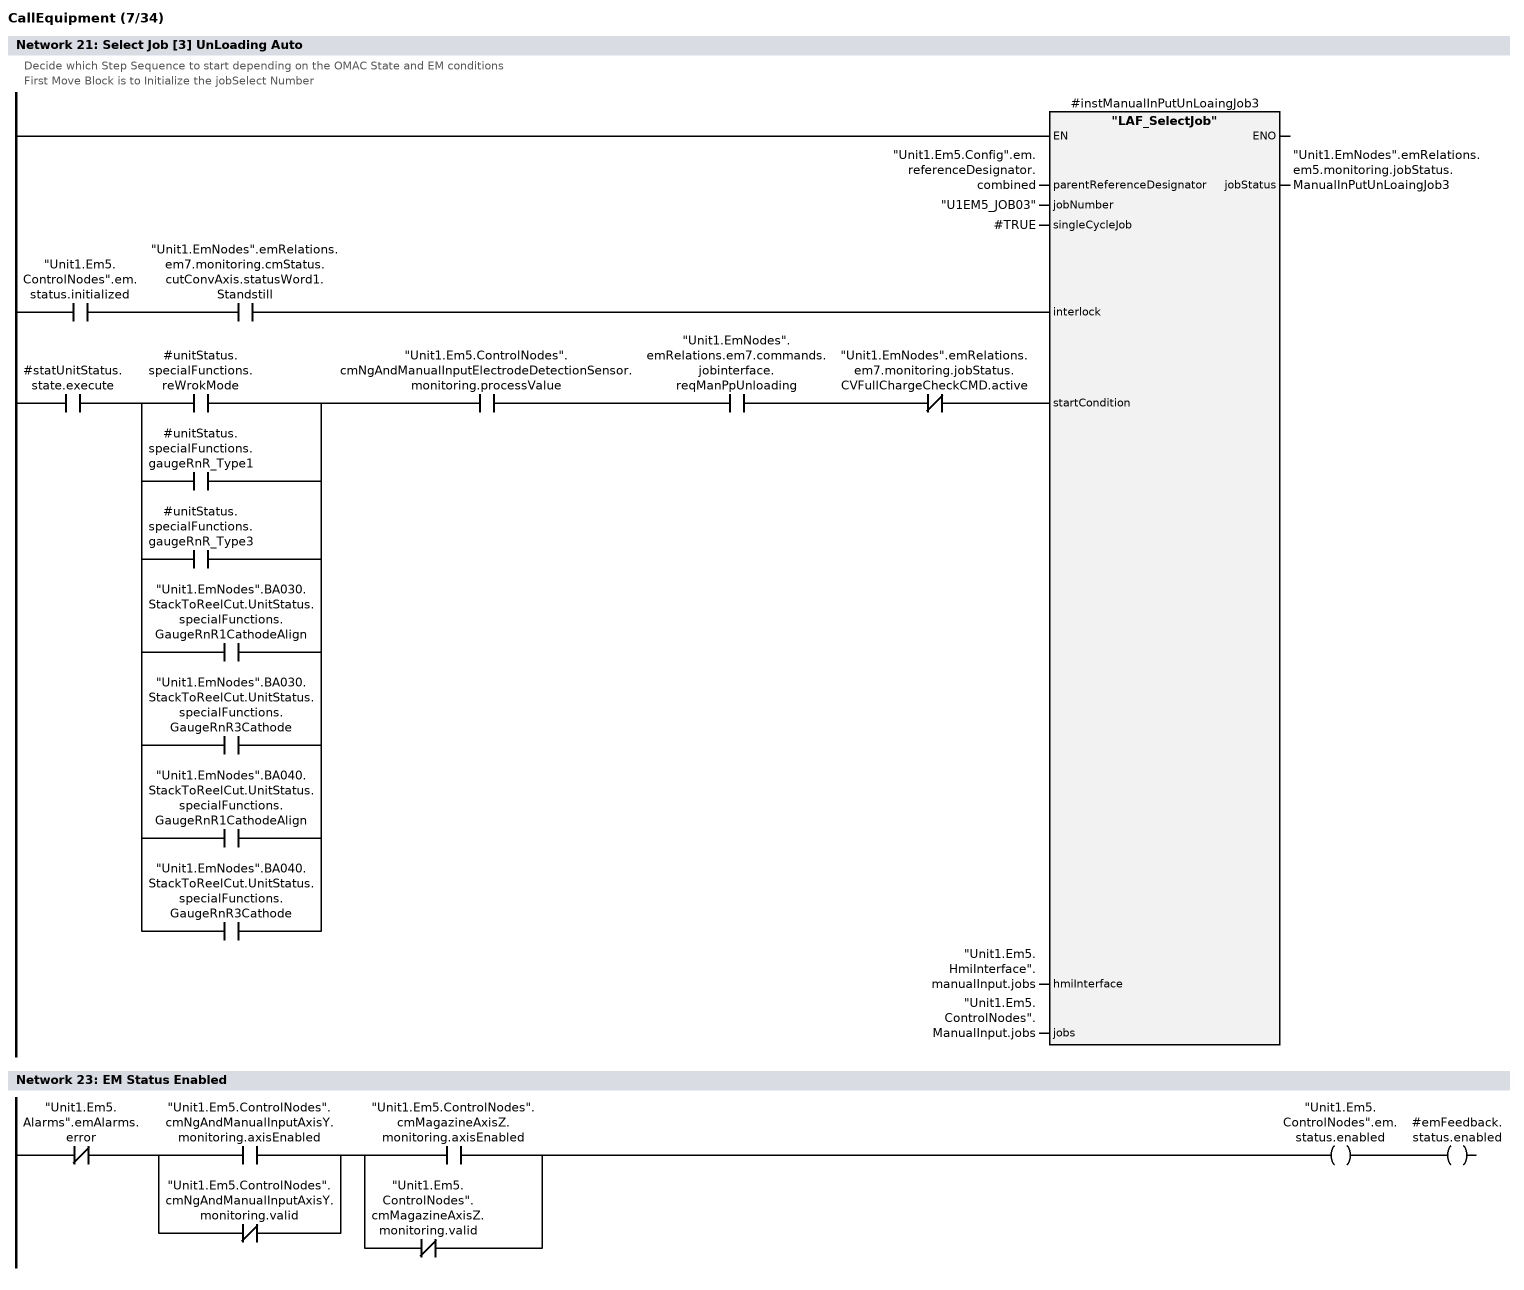
   RUNG wire#powerrail
      #instManualInPutUnLoaingJob3(interlock := wire#w1, startCondition := wire#w4, parentReferenceDesignator := "Unit1.Em5.Config".em.referenceDesignator.combined, jobNumber := "U1EM5_JOB03", singleCycleJob := #TRUE, hmiInterface := "Unit1.Em5.HmiInterface".manualInput.jobs, jobs := "Unit1.Em5.ControlNodes".ManualInput.jobs, jobStatus => "Unit1.EmNodes".emRelations.em5.monitoring.jobStatus.ManualInPutUnLoaingJob3)
   END_RUNG
   RUNG wire#powerrail
      Contact( "Unit1.Em5.ControlNodes".em.status.initialized )
      Contact( "Unit1.EmNodes".emRelations.em7.monitoring.cmStatus.cutConvAxis.statusWord1.Standstill )
   END_RUNG wire#w1
   RUNG wire#powerrail
      Contact( #statUnitStatus.state.execute )
      wire#w2
      Contact( #unitStatus.specialFunctions.reWrokMode )
      wire#w3
      Contact( "Unit1.Em5.ControlNodes".cmNgAndManualInputElectrodeDetectionSensor.monitoring.processValue )
      Contact( "Unit1.EmNodes".emRelations.em7.commands.jobinterface.reqManPpUnloading )
      I_Contact( "Unit1.EmNodes".emRelations.em7.monitoring.jobStatus.CVFullChargeCheckCMD.active )
   END_RUNG wire#w4
   RUNG wire#w2
      Contact( #unitStatus.specialFunctions.gaugeRnR_Type1 )
   END_RUNG wire#w3
   RUNG wire#w2
      Contact( #unitStatus.specialFunctions.gaugeRnR_Type3 )
   END_RUNG wire#w3
   RUNG wire#w2
      Contact( "Unit1.EmNodes".BA030.StackToReelCut.UnitStatus.specialFunctions.GaugeRnR1CathodeAlign )
   END_RUNG wire#w3
   RUNG wire#w2
      Contact( "Unit1.EmNodes".BA030.StackToReelCut.UnitStatus.specialFunctions.GaugeRnR3Cathode )
   END_RUNG wire#w3
   RUNG wire#w2
      Contact( "Unit1.EmNodes".BA040.StackToReelCut.UnitStatus.specialFunctions.GaugeRnR1CathodeAlign )
   END_RUNG wire#w3
   RUNG wire#w2
      Contact( "Unit1.EmNodes".BA040.StackToReelCut.UnitStatus.specialFunctions.GaugeRnR3Cathode )
   END_RUNG wire#w3
   // the same network as SCL:
   #instManualInPutUnLoaingJob3(parentReferenceDesignator := "Unit1.Em5.Config".em.referenceDesignator.combined,   // "LAF_SelectJob"
                           jobNumber := "U1EM5_JOB03",
                           singleCycleJob := #TRUE,
                           interlock := "Unit1.Em5.ControlNodes".em.status.initialized AND "Unit1.EmNodes".emRelations.em7.monitoring.cmStatus.cutConvAxis.statusWord1.Standstill,
                           startCondition := #statUnitStatus.state.execute AND (#unitStatus.specialFunctions.reWrokMode OR #unitStatus.specialFunctions.gaugeRnR_Type1 OR #unitStatus.specialFunctions.gaugeRnR_Type3 OR "Unit1.EmNodes".BA030.StackToReelCut.UnitStatus.specialFunctions.GaugeRnR1CathodeAlign OR "Unit1.EmNodes".BA030.StackToReelCut.UnitStatus.specialFunctions.GaugeRnR3Cathode OR "Unit1.EmNodes".BA040.StackToReelCut.UnitStatus.specialFunctions.GaugeRnR1CathodeAlign OR "Unit1.EmNodes".BA040.StackToReelCut.UnitStatus.specialFunctions.GaugeRnR3Cathode) AND "Unit1.Em5.ControlNodes".cmNgAndManualInputElectrodeDetectionSensor.monitoring.processValue AND "Unit1.EmNodes".emRelations.em7.commands.jobinterface.reqManPpUnloading AND NOT "Unit1.EmNodes".emRelations.em7.monitoring.jobStatus.CVFullChargeCheckCMD.active,
                           hmiInterface := "Unit1.Em5.HmiInterface".manualInput.jobs,
                           jobs := "Unit1.Em5.ControlNodes".ManualInput.jobs,
                           jobStatus => "Unit1.EmNodes".emRelations.em5.monitoring.jobStatus.ManualInPutUnLoaingJob3);
END_REGION

REGION Network 22: Select Job Working Done
END_REGION

REGION Network 23: EM Status Enabled
   RUNG wire#powerrail
      I_Contact( "Unit1.Em5.Alarms".emAlarms.error )
      wire#w1
      Contact( "Unit1.Em5.ControlNodes".cmNgAndManualInputAxisY.monitoring.axisEnabled )
      wire#w2
      Contact( "Unit1.Em5.ControlNodes".cmMagazineAxisZ.monitoring.axisEnabled )
      wire#w3
      Coil( "Unit1.Em5.ControlNodes".em.status.enabled )
      Coil( #emFeedback.status.enabled )
   END_RUNG
   RUNG wire#w1
      I_Contact( "Unit1.Em5.ControlNodes".cmNgAndManualInputAxisY.monitoring.valid )
   END_RUNG wire#w2
   RUNG wire#w2
      I_Contact( "Unit1.Em5.ControlNodes".cmMagazineAxisZ.monitoring.valid )
   END_RUNG wire#w3
   // the same network as SCL:
   "Unit1.Em5.ControlNodes".em.status.enabled := NOT "Unit1.Em5.Alarms".emAlarms.error AND ("Unit1.Em5.ControlNodes".cmNgAndManualInputAxisY.monitoring.axisEnabled OR NOT "Unit1.Em5.ControlNodes".cmNgAndManualInputAxisY.monitoring.valid) AND ("Unit1.Em5.ControlNodes".cmMagazineAxisZ.monitoring.axisEnabled OR NOT "Unit1.Em5.ControlNodes".cmMagazineAxisZ.monitoring.valid);
   #emFeedback.status.enabled := "Unit1.Em5.ControlNodes".em.status.enabled;
END_REGION

REGION Network 24: EM Status initialized
   // Set em to initialized here. Usually this is done when the initialization job is completed.
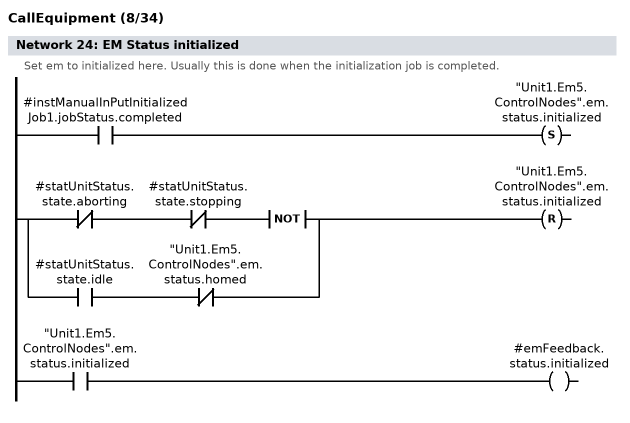
   RUNG wire#powerrail
      Contact( #instManualInPutInitializedJob1.jobStatus.completed )
      S_Coil( "Unit1.Em5.ControlNodes".em.status.initialized )
   END_RUNG
   RUNG wire#powerrail
      I_Contact( #statUnitStatus.state.aborting )
      I_Contact( #statUnitStatus.state.stopping )
      Not()
      wire#w1
      R_Coil( "Unit1.Em5.ControlNodes".em.status.initialized )
   END_RUNG
   RUNG wire#powerrail
      Contact( #statUnitStatus.state.idle )
      I_Contact( "Unit1.Em5.ControlNodes".em.status.homed )
   END_RUNG wire#w1
   RUNG wire#powerrail
      Contact( "Unit1.Em5.ControlNodes".em.status.initialized )
      Coil( #emFeedback.status.initialized )
   END_RUNG
   // the same network as SCL:
   IF #instManualInPutInitializedJob1.jobStatus.completed THEN
       "Unit1.Em5.ControlNodes".em.status.initialized := TRUE;
   END_IF;
   IF NOT (NOT #statUnitStatus.state.aborting AND NOT #statUnitStatus.state.stopping) OR (#statUnitStatus.state.idle AND NOT "Unit1.Em5.ControlNodes".em.status.homed) THEN
       "Unit1.Em5.ControlNodes".em.status.initialized := FALSE;
   END_IF;
   #emFeedback.status.initialized := "Unit1.Em5.ControlNodes".em.status.initialized;
END_REGION

REGION Network 25: EM Status Homed
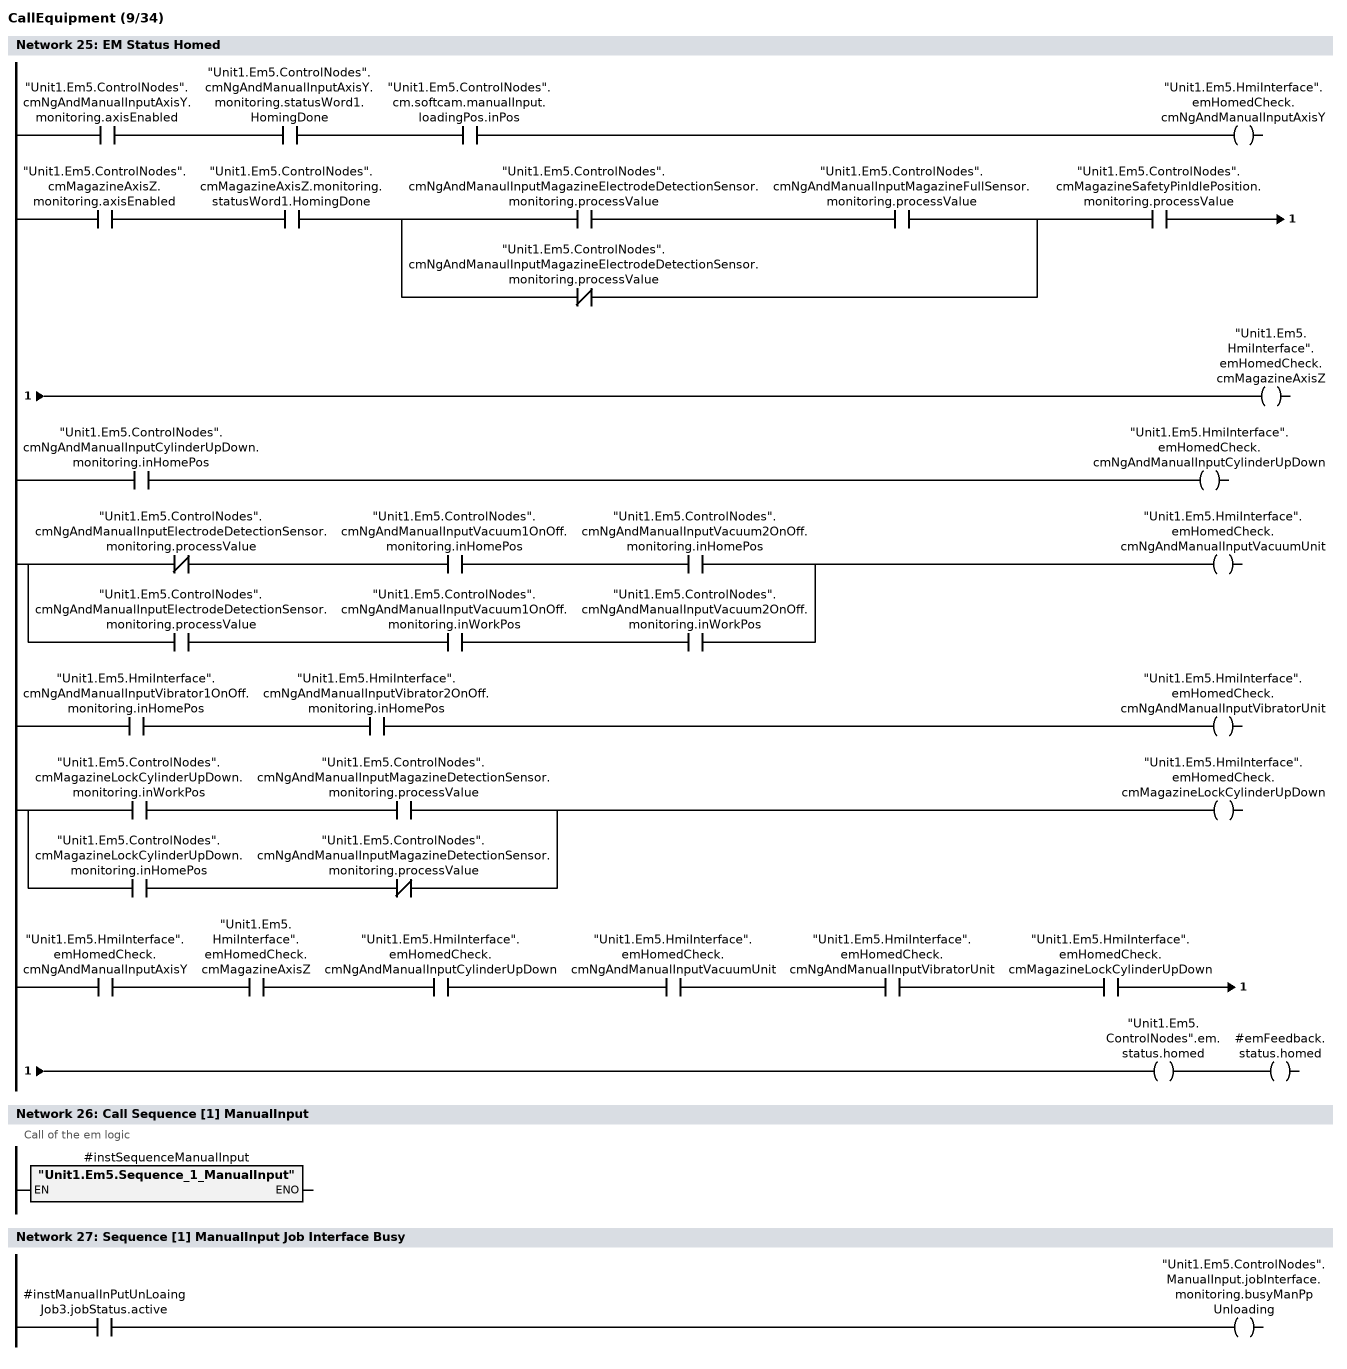
   RUNG wire#powerrail
      Contact( "Unit1.Em5.ControlNodes".cmNgAndManualInputAxisY.monitoring.axisEnabled )
      Contact( "Unit1.Em5.ControlNodes".cmNgAndManualInputAxisY.monitoring.statusWord1.HomingDone )
      Contact( "Unit1.Em5.ControlNodes".cm.softcam.manualInput.loadingPos.inPos )
      Coil( "Unit1.Em5.HmiInterface".emHomedCheck.cmNgAndManualInputAxisY )
   END_RUNG
   RUNG wire#powerrail
      Contact( "Unit1.Em5.ControlNodes".cmMagazineAxisZ.monitoring.axisEnabled )
      Contact( "Unit1.Em5.ControlNodes".cmMagazineAxisZ.monitoring.statusWord1.HomingDone )
      wire#w1
      Contact( "Unit1.Em5.ControlNodes".cmNgAndManaulInputMagazineElectrodeDetectionSensor.monitoring.processValue )
      Contact( "Unit1.Em5.ControlNodes".cmNgAndManualInputMagazineFullSensor.monitoring.processValue )
      wire#w2
      Contact( "Unit1.Em5.ControlNodes".cmMagazineSafetyPinIdlePosition.monitoring.processValue )
      Coil( "Unit1.Em5.HmiInterface".emHomedCheck.cmMagazineAxisZ )
   END_RUNG
   RUNG wire#w1
      I_Contact( "Unit1.Em5.ControlNodes".cmNgAndManaulInputMagazineElectrodeDetectionSensor.monitoring.processValue )
   END_RUNG wire#w2
   RUNG wire#powerrail
      Contact( "Unit1.Em5.ControlNodes".cmNgAndManualInputCylinderUpDown.monitoring.inHomePos )
      Coil( "Unit1.Em5.HmiInterface".emHomedCheck.cmNgAndManualInputCylinderUpDown )
   END_RUNG
   RUNG wire#powerrail
      I_Contact( "Unit1.Em5.ControlNodes".cmNgAndManualInputElectrodeDetectionSensor.monitoring.processValue )
      Contact( "Unit1.Em5.ControlNodes".cmNgAndManualInputVacuum1OnOff.monitoring.inHomePos )
      Contact( "Unit1.Em5.ControlNodes".cmNgAndManualInputVacuum2OnOff.monitoring.inHomePos )
      wire#w3
      Coil( "Unit1.Em5.HmiInterface".emHomedCheck.cmNgAndManualInputVacuumUnit )
   END_RUNG
   RUNG wire#powerrail
      Contact( "Unit1.Em5.ControlNodes".cmNgAndManualInputElectrodeDetectionSensor.monitoring.processValue )
      Contact( "Unit1.Em5.ControlNodes".cmNgAndManualInputVacuum1OnOff.monitoring.inWorkPos )
      Contact( "Unit1.Em5.ControlNodes".cmNgAndManualInputVacuum2OnOff.monitoring.inWorkPos )
   END_RUNG wire#w3
   RUNG wire#powerrail
      Contact( "Unit1.Em5.HmiInterface".cmNgAndManualInputVibrator1OnOff.monitoring.inHomePos )
      Contact( "Unit1.Em5.HmiInterface".cmNgAndManualInputVibrator2OnOff.monitoring.inHomePos )
      Coil( "Unit1.Em5.HmiInterface".emHomedCheck.cmNgAndManualInputVibratorUnit )
   END_RUNG
   RUNG wire#powerrail
      Contact( "Unit1.Em5.ControlNodes".cmMagazineLockCylinderUpDown.monitoring.inWorkPos )
      Contact( "Unit1.Em5.ControlNodes".cmNgAndManualInputMagazineDetectionSensor.monitoring.processValue )
      wire#w4
      Coil( "Unit1.Em5.HmiInterface".emHomedCheck.cmMagazineLockCylinderUpDown )
   END_RUNG
   RUNG wire#powerrail
      Contact( "Unit1.Em5.ControlNodes".cmMagazineLockCylinderUpDown.monitoring.inHomePos )
      I_Contact( "Unit1.Em5.ControlNodes".cmNgAndManualInputMagazineDetectionSensor.monitoring.processValue )
   END_RUNG wire#w4
   RUNG wire#powerrail
      Contact( "Unit1.Em5.HmiInterface".emHomedCheck.cmNgAndManualInputAxisY )
      Contact( "Unit1.Em5.HmiInterface".emHomedCheck.cmMagazineAxisZ )
      Contact( "Unit1.Em5.HmiInterface".emHomedCheck.cmNgAndManualInputCylinderUpDown )
      Contact( "Unit1.Em5.HmiInterface".emHomedCheck.cmNgAndManualInputVacuumUnit )
      Contact( "Unit1.Em5.HmiInterface".emHomedCheck.cmNgAndManualInputVibratorUnit )
      Contact( "Unit1.Em5.HmiInterface".emHomedCheck.cmMagazineLockCylinderUpDown )
      Coil( "Unit1.Em5.ControlNodes".em.status.homed )
      Coil( #emFeedback.status.homed )
   END_RUNG
   // the same network as SCL:
   "Unit1.Em5.HmiInterface".emHomedCheck.cmNgAndManualInputAxisY := "Unit1.Em5.ControlNodes".cmNgAndManualInputAxisY.monitoring.axisEnabled AND "Unit1.Em5.ControlNodes".cmNgAndManualInputAxisY.monitoring.statusWord1.HomingDone AND "Unit1.Em5.ControlNodes".cm.softcam.manualInput.loadingPos.inPos;
   "Unit1.Em5.HmiInterface".emHomedCheck.cmMagazineAxisZ := "Unit1.Em5.ControlNodes".cmMagazineAxisZ.monitoring.axisEnabled AND "Unit1.Em5.ControlNodes".cmMagazineAxisZ.monitoring.statusWord1.HomingDone AND (("Unit1.Em5.ControlNodes".cmNgAndManaulInputMagazineElectrodeDetectionSensor.monitoring.processValue AND "Unit1.Em5.ControlNodes".cmNgAndManualInputMagazineFullSensor.monitoring.processValue) OR NOT "Unit1.Em5.ControlNodes".cmNgAndManaulInputMagazineElectrodeDetectionSensor.monitoring.processValue) AND "Unit1.Em5.ControlNodes".cmMagazineSafetyPinIdlePosition.monitoring.processValue;
   "Unit1.Em5.HmiInterface".emHomedCheck.cmNgAndManualInputCylinderUpDown := "Unit1.Em5.ControlNodes".cmNgAndManualInputCylinderUpDown.monitoring.inHomePos;
   "Unit1.Em5.HmiInterface".emHomedCheck.cmNgAndManualInputVacuumUnit := (NOT "Unit1.Em5.ControlNodes".cmNgAndManualInputElectrodeDetectionSensor.monitoring.processValue AND "Unit1.Em5.ControlNodes".cmNgAndManualInputVacuum1OnOff.monitoring.inHomePos AND "Unit1.Em5.ControlNodes".cmNgAndManualInputVacuum2OnOff.monitoring.inHomePos) OR ("Unit1.Em5.ControlNodes".cmNgAndManualInputElectrodeDetectionSensor.monitoring.processValue AND "Unit1.Em5.ControlNodes".cmNgAndManualInputVacuum1OnOff.monitoring.inWorkPos AND "Unit1.Em5.ControlNodes".cmNgAndManualInputVacuum2OnOff.monitoring.inWorkPos);
   "Unit1.Em5.HmiInterface".emHomedCheck.cmNgAndManualInputVibratorUnit := "Unit1.Em5.HmiInterface".cmNgAndManualInputVibrator1OnOff.monitoring.inHomePos AND "Unit1.Em5.HmiInterface".cmNgAndManualInputVibrator2OnOff.monitoring.inHomePos;
   "Unit1.Em5.HmiInterface".emHomedCheck.cmMagazineLockCylinderUpDown := ("Unit1.Em5.ControlNodes".cmMagazineLockCylinderUpDown.monitoring.inWorkPos AND "Unit1.Em5.ControlNodes".cmNgAndManualInputMagazineDetectionSensor.monitoring.processValue) OR ("Unit1.Em5.ControlNodes".cmMagazineLockCylinderUpDown.monitoring.inHomePos AND NOT "Unit1.Em5.ControlNodes".cmNgAndManualInputMagazineDetectionSensor.monitoring.processValue);
   "Unit1.Em5.ControlNodes".em.status.homed := "Unit1.Em5.HmiInterface".emHomedCheck.cmNgAndManualInputAxisY AND "Unit1.Em5.HmiInterface".emHomedCheck.cmMagazineAxisZ AND "Unit1.Em5.HmiInterface".emHomedCheck.cmNgAndManualInputCylinderUpDown AND "Unit1.Em5.HmiInterface".emHomedCheck.cmNgAndManualInputVacuumUnit AND "Unit1.Em5.HmiInterface".emHomedCheck.cmNgAndManualInputVibratorUnit AND "Unit1.Em5.HmiInterface".emHomedCheck.cmMagazineLockCylinderUpDown;
   #emFeedback.status.homed := "Unit1.Em5.ControlNodes".em.status.homed;
END_REGION

REGION Network 26: Call Sequence [1] ManualInput
   // Call of the em logic
   RUNG wire#powerrail
      #instSequenceManualInput()
   END_RUNG
   // the same network as SCL:
   #instSequenceManualInput();   // "Unit1.Em5.Sequence_1_ManualInput"
END_REGION

REGION Network 27: Sequence [1] ManualInput Job Interface Busy
   RUNG wire#powerrail
      Contact( #instManualInPutUnLoaingJob3.jobStatus.active )
      Coil( "Unit1.Em5.ControlNodes".ManualInput.jobInterface.monitoring.busyManPpUnloading )
   END_RUNG
   // the same network as SCL:
   "Unit1.Em5.ControlNodes".ManualInput.jobInterface.monitoring.busyManPpUnloading := #instManualInPutUnLoaingJob3.jobStatus.active;
END_REGION

REGION Network 28: Sequence [1] ManualInput Job Interface Done
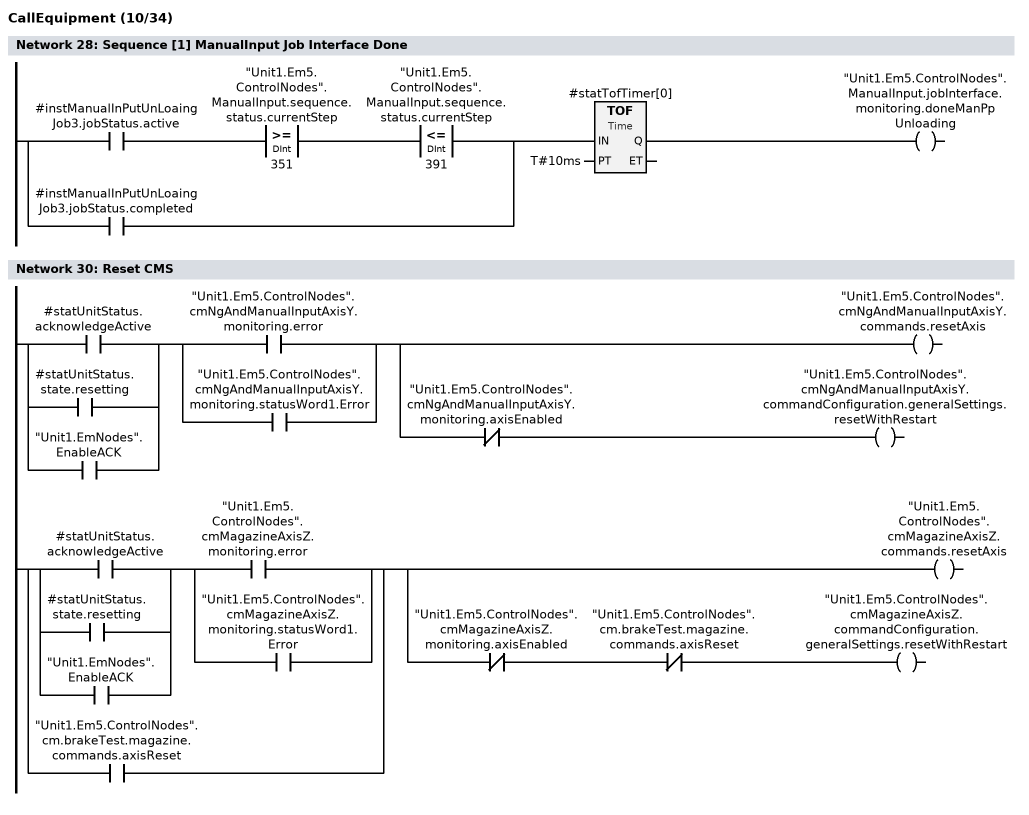
   RUNG wire#powerrail
      Contact( #instManualInPutUnLoaingJob3.jobStatus.active )
      { S7_Templates := "SrcType := DInt" } GE_Contact(in1 := "Unit1.Em5.ControlNodes".ManualInput.sequence.status.currentStep, in2 := 351)
      { S7_Templates := "SrcType := DInt" } LE_Contact(in1 := "Unit1.Em5.ControlNodes".ManualInput.sequence.status.currentStep, in2 := 391)
      wire#w1
      { S7_Templates := "time_type := Time" } #statTofTimer[0].TOF(pt := T#10ms, et =>)
      Coil( "Unit1.Em5.ControlNodes".ManualInput.jobInterface.monitoring.doneManPpUnloading )
   END_RUNG
   RUNG wire#powerrail
      Contact( #instManualInPutUnLoaingJob3.jobStatus.completed )
   END_RUNG wire#w1
   // the same network as SCL:
   #statTofTimer[0].TOF(IN := (#instManualInPutUnLoaingJob3.jobStatus.active AND ("Unit1.Em5.ControlNodes".ManualInput.sequence.status.currentStep >= 351) AND ("Unit1.Em5.ControlNodes".ManualInput.sequence.status.currentStep <= 391)) OR #instManualInPutUnLoaingJob3.jobStatus.completed,
                        PT := T#10ms);
   "Unit1.Em5.ControlNodes".ManualInput.jobInterface.monitoring.doneManPpUnloading := #statTofTimer[0].Q;
END_REGION

REGION Network 29: ******************** Control Modules (Axis) ********************
   // Call control modules that are actuators after the em logic (jobs and sequence), so that the latest commands are applied to the actuators.
END_REGION

REGION Network 30: Reset CMS
   RUNG wire#powerrail
      Contact( #statUnitStatus.acknowledgeActive )
      wire#w1
      Contact( "Unit1.Em5.ControlNodes".cmNgAndManualInputAxisY.monitoring.error )
      wire#w2
      Coil( "Unit1.Em5.ControlNodes".cmNgAndManualInputAxisY.commands.resetAxis )
   END_RUNG
   RUNG wire#powerrail
      Contact( #statUnitStatus.state.resetting )
   END_RUNG wire#w1
   RUNG wire#powerrail
      Contact( "Unit1.EmNodes".EnableACK )
   END_RUNG wire#w1
   RUNG wire#w1
      Contact( "Unit1.Em5.ControlNodes".cmNgAndManualInputAxisY.monitoring.statusWord1.Error )
   END_RUNG wire#w2
   RUNG wire#w2
      I_Contact( "Unit1.Em5.ControlNodes".cmNgAndManualInputAxisY.monitoring.axisEnabled )
      Coil( "Unit1.Em5.ControlNodes".cmNgAndManualInputAxisY.commandConfiguration.generalSettings.resetWithRestart )
   END_RUNG
   RUNG wire#powerrail
      Contact( #statUnitStatus.acknowledgeActive )
      wire#w3
      Contact( "Unit1.Em5.ControlNodes".cmMagazineAxisZ.monitoring.error )
      wire#w4
      Coil( "Unit1.Em5.ControlNodes".cmMagazineAxisZ.commands.resetAxis )
   END_RUNG
   RUNG wire#powerrail
      Contact( #statUnitStatus.state.resetting )
   END_RUNG wire#w3
   RUNG wire#powerrail
      Contact( "Unit1.EmNodes".EnableACK )
   END_RUNG wire#w3
   RUNG wire#w3
      Contact( "Unit1.Em5.ControlNodes".cmMagazineAxisZ.monitoring.statusWord1.Error )
   END_RUNG wire#w4
   RUNG wire#powerrail
      Contact( "Unit1.Em5.ControlNodes".cm.brakeTest.magazine.commands.axisReset )
   END_RUNG wire#w4
   RUNG wire#w4
      I_Contact( "Unit1.Em5.ControlNodes".cmMagazineAxisZ.monitoring.axisEnabled )
      I_Contact( "Unit1.Em5.ControlNodes".cm.brakeTest.magazine.commands.axisReset )
      Coil( "Unit1.Em5.ControlNodes".cmMagazineAxisZ.commandConfiguration.generalSettings.resetWithRestart )
   END_RUNG
   // the same network as SCL:
   "Unit1.Em5.ControlNodes".cmNgAndManualInputAxisY.commands.resetAxis := (#statUnitStatus.acknowledgeActive OR #statUnitStatus.state.resetting OR "Unit1.EmNodes".EnableACK) AND ("Unit1.Em5.ControlNodes".cmNgAndManualInputAxisY.monitoring.error OR "Unit1.Em5.ControlNodes".cmNgAndManualInputAxisY.monitoring.statusWord1.Error);
   "Unit1.Em5.ControlNodes".cmNgAndManualInputAxisY.commandConfiguration.generalSettings.resetWithRestart := "Unit1.Em5.ControlNodes".cmNgAndManualInputAxisY.commands.resetAxis AND NOT "Unit1.Em5.ControlNodes".cmNgAndManualInputAxisY.monitoring.axisEnabled;
   "Unit1.Em5.ControlNodes".cmMagazineAxisZ.commands.resetAxis := ((#statUnitStatus.acknowledgeActive OR #statUnitStatus.state.resetting OR "Unit1.EmNodes".EnableACK) AND ("Unit1.Em5.ControlNodes".cmMagazineAxisZ.monitoring.error OR "Unit1.Em5.ControlNodes".cmMagazineAxisZ.monitoring.statusWord1.Error)) OR "Unit1.Em5.ControlNodes".cm.brakeTest.magazine.commands.axisReset;
   "Unit1.Em5.ControlNodes".cmMagazineAxisZ.commandConfiguration.generalSettings.resetWithRestart := "Unit1.Em5.ControlNodes".cmMagazineAxisZ.commands.resetAxis AND NOT "Unit1.Em5.ControlNodes".cmMagazineAxisZ.monitoring.axisEnabled AND NOT "Unit1.Em5.ControlNodes".cm.brakeTest.magazine.commands.axisReset;
END_REGION

REGION Network 31: Enable/Disable CMs
   // Enable the axis during the resetting state and disable the axis during the aborting state.
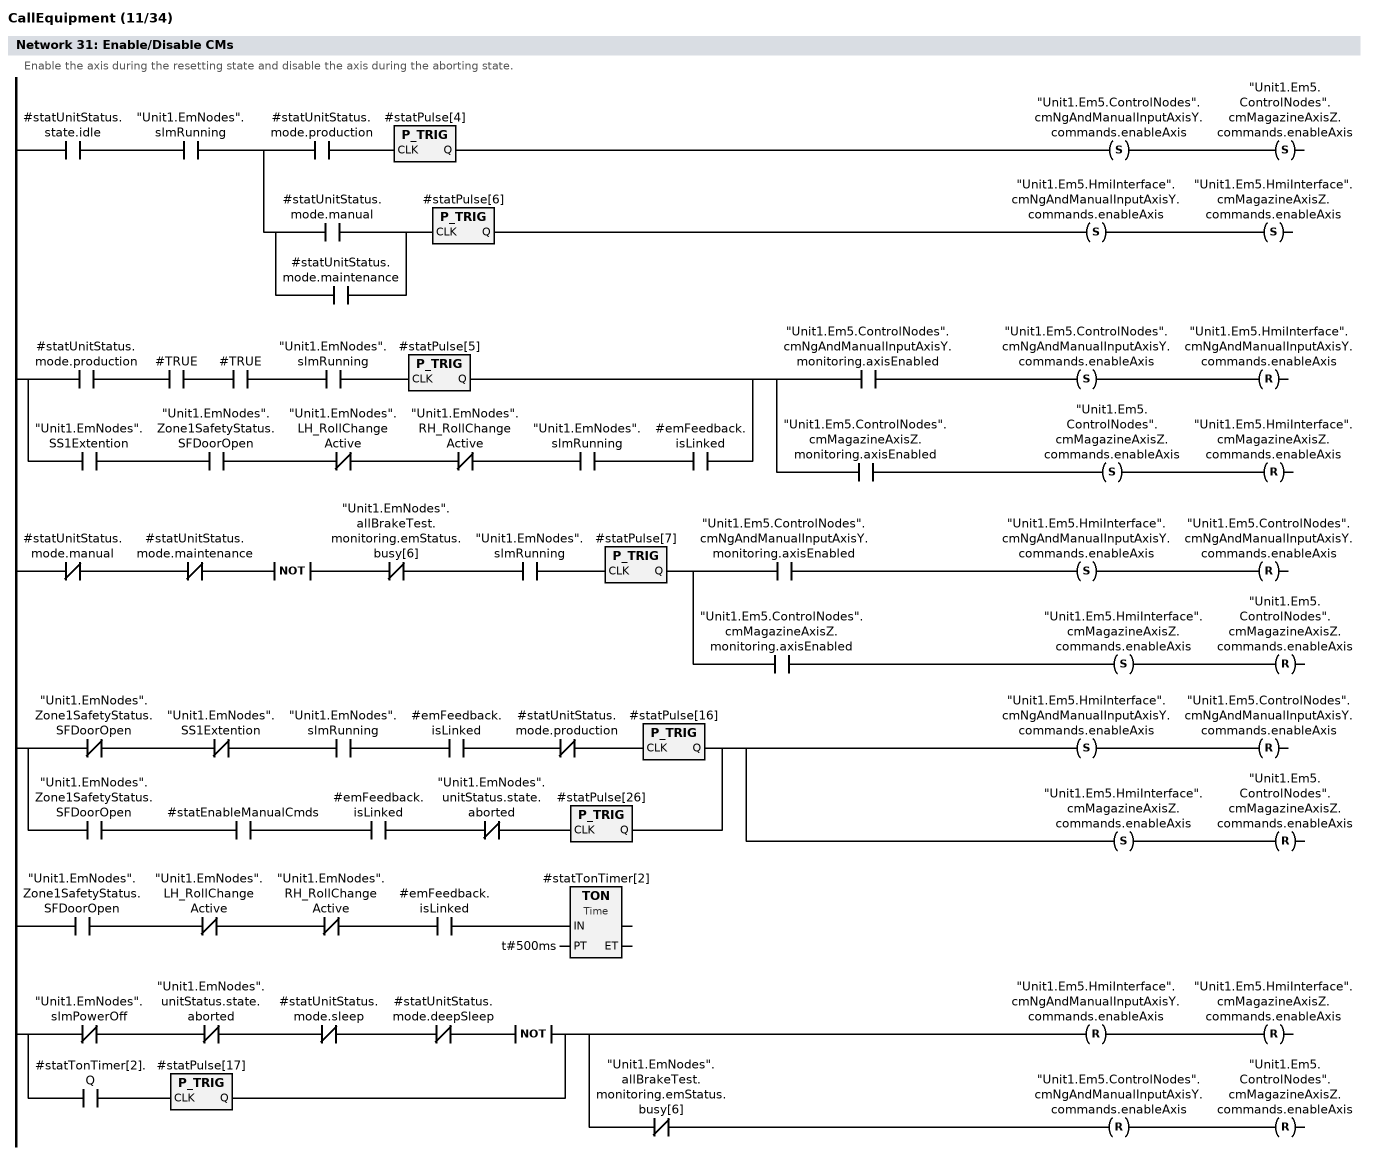
   RUNG wire#powerrail
      Contact( #statUnitStatus.state.idle )
      Contact( "Unit1.EmNodes".slmRunning )
      wire#w1
      Contact( #statUnitStatus.mode.production )
      P_Trig( #statPulse[4] )
      S_Coil( "Unit1.Em5.ControlNodes".cmNgAndManualInputAxisY.commands.enableAxis )
      S_Coil( "Unit1.Em5.ControlNodes".cmMagazineAxisZ.commands.enableAxis )
   END_RUNG
   RUNG wire#w1
      Contact( #statUnitStatus.mode.manual )
      wire#w2
      P_Trig( #statPulse[6] )
      S_Coil( "Unit1.Em5.HmiInterface".cmNgAndManualInputAxisY.commands.enableAxis )
      S_Coil( "Unit1.Em5.HmiInterface".cmMagazineAxisZ.commands.enableAxis )
   END_RUNG
   RUNG wire#w1
      Contact( #statUnitStatus.mode.maintenance )
   END_RUNG wire#w2
   RUNG wire#powerrail
      Contact( #statUnitStatus.mode.production )
      Contact( #TRUE )
      Contact( #TRUE )
      Contact( "Unit1.EmNodes".slmRunning )
      P_Trig( #statPulse[5] )
      wire#w3
      Contact( "Unit1.Em5.ControlNodes".cmNgAndManualInputAxisY.monitoring.axisEnabled )
      S_Coil( "Unit1.Em5.ControlNodes".cmNgAndManualInputAxisY.commands.enableAxis )
      R_Coil( "Unit1.Em5.HmiInterface".cmNgAndManualInputAxisY.commands.enableAxis )
   END_RUNG
   RUNG wire#powerrail
      Contact( "Unit1.EmNodes".SS1Extention )
      Contact( "Unit1.EmNodes".Zone1SafetyStatus.SFDoorOpen )
      I_Contact( "Unit1.EmNodes".LH_RollChangeActive )
      I_Contact( "Unit1.EmNodes".RH_RollChangeActive )
      Contact( "Unit1.EmNodes".slmRunning )
      Contact( #emFeedback.isLinked )
   END_RUNG wire#w3
   RUNG wire#w3
      Contact( "Unit1.Em5.ControlNodes".cmMagazineAxisZ.monitoring.axisEnabled )
      S_Coil( "Unit1.Em5.ControlNodes".cmMagazineAxisZ.commands.enableAxis )
      R_Coil( "Unit1.Em5.HmiInterface".cmMagazineAxisZ.commands.enableAxis )
   END_RUNG
   RUNG wire#powerrail
      I_Contact( #statUnitStatus.mode.manual )
      I_Contact( #statUnitStatus.mode.maintenance )
      Not()
      I_Contact( "Unit1.EmNodes".allBrakeTest.monitoring.emStatus.busy[6] )
      Contact( "Unit1.EmNodes".slmRunning )
      P_Trig( #statPulse[7] )
      wire#w4
      Contact( "Unit1.Em5.ControlNodes".cmNgAndManualInputAxisY.monitoring.axisEnabled )
      S_Coil( "Unit1.Em5.HmiInterface".cmNgAndManualInputAxisY.commands.enableAxis )
      R_Coil( "Unit1.Em5.ControlNodes".cmNgAndManualInputAxisY.commands.enableAxis )
   END_RUNG
   RUNG wire#w4
      Contact( "Unit1.Em5.ControlNodes".cmMagazineAxisZ.monitoring.axisEnabled )
      S_Coil( "Unit1.Em5.HmiInterface".cmMagazineAxisZ.commands.enableAxis )
      R_Coil( "Unit1.Em5.ControlNodes".cmMagazineAxisZ.commands.enableAxis )
   END_RUNG
   RUNG wire#powerrail
      I_Contact( "Unit1.EmNodes".Zone1SafetyStatus.SFDoorOpen )
      I_Contact( "Unit1.EmNodes".SS1Extention )
      Contact( "Unit1.EmNodes".slmRunning )
      Contact( #emFeedback.isLinked )
      I_Contact( #statUnitStatus.mode.production )
      P_Trig( #statPulse[16] )
      wire#w5
      S_Coil( "Unit1.Em5.HmiInterface".cmNgAndManualInputAxisY.commands.enableAxis )
      R_Coil( "Unit1.Em5.ControlNodes".cmNgAndManualInputAxisY.commands.enableAxis )
   END_RUNG
   RUNG wire#powerrail
      Contact( "Unit1.EmNodes".Zone1SafetyStatus.SFDoorOpen )
      Contact( #statEnableManualCmds )
      Contact( #emFeedback.isLinked )
      I_Contact( "Unit1.EmNodes".unitStatus.state.aborted )
      P_Trig( #statPulse[26] )
   END_RUNG wire#w5
   RUNG wire#w5
      S_Coil( "Unit1.Em5.HmiInterface".cmMagazineAxisZ.commands.enableAxis )
      R_Coil( "Unit1.Em5.ControlNodes".cmMagazineAxisZ.commands.enableAxis )
   END_RUNG
   RUNG wire#powerrail
      Contact( "Unit1.EmNodes".Zone1SafetyStatus.SFDoorOpen )
      I_Contact( "Unit1.EmNodes".LH_RollChangeActive )
      I_Contact( "Unit1.EmNodes".RH_RollChangeActive )
      Contact( #emFeedback.isLinked )
      { S7_Templates := "time_type := Time" } #statTonTimer[2].TON(pt := t#500ms, et =>)
   END_RUNG
   RUNG wire#powerrail
      I_Contact( "Unit1.EmNodes".slmPowerOff )
      I_Contact( "Unit1.EmNodes".unitStatus.state.aborted )
      I_Contact( #statUnitStatus.mode.sleep )
      I_Contact( #statUnitStatus.mode.deepSleep )
      Not()
      wire#w6
      R_Coil( "Unit1.Em5.HmiInterface".cmNgAndManualInputAxisY.commands.enableAxis )
      R_Coil( "Unit1.Em5.HmiInterface".cmMagazineAxisZ.commands.enableAxis )
   END_RUNG
   RUNG wire#powerrail
      Contact( #statTonTimer[2].Q )
      P_Trig( #statPulse[17] )
   END_RUNG wire#w6
   RUNG wire#w6
      I_Contact( "Unit1.EmNodes".allBrakeTest.monitoring.emStatus.busy[6] )
      R_Coil( "Unit1.Em5.ControlNodes".cmNgAndManualInputAxisY.commands.enableAxis )
      R_Coil( "Unit1.Em5.ControlNodes".cmMagazineAxisZ.commands.enableAxis )
   END_RUNG
   // the same network as SCL:
   #_w1 := #statUnitStatus.state.idle AND "Unit1.EmNodes".slmRunning;
   #_w2 := #_w1 AND #statUnitStatus.mode.production;
   #_w3 := #_w2 AND NOT #statPulse[4];   // rising edge
   #statPulse[4] := #_w2;
   IF #_w3 THEN
       "Unit1.Em5.ControlNodes".cmNgAndManualInputAxisY.commands.enableAxis := TRUE;
       "Unit1.Em5.ControlNodes".cmMagazineAxisZ.commands.enableAxis := TRUE;
   END_IF;
   #_w4 := #_w1 AND (#statUnitStatus.mode.manual OR #statUnitStatus.mode.maintenance);
   #_w5 := #_w4 AND NOT #statPulse[6];   // rising edge
   #statPulse[6] := #_w4;
   IF #_w5 THEN
       "Unit1.Em5.HmiInterface".cmNgAndManualInputAxisY.commands.enableAxis := TRUE;
       "Unit1.Em5.HmiInterface".cmMagazineAxisZ.commands.enableAxis := TRUE;
   END_IF;
   #_w6 := #statUnitStatus.mode.production AND #TRUE AND #TRUE AND "Unit1.EmNodes".slmRunning;
   #_w7 := #_w6 AND NOT #statPulse[5];   // rising edge
   #statPulse[5] := #_w6;
   #_w8 := #_w7 OR ("Unit1.EmNodes".SS1Extention AND "Unit1.EmNodes".Zone1SafetyStatus.SFDoorOpen AND NOT "Unit1.EmNodes".LH_RollChangeActive AND NOT "Unit1.EmNodes".RH_RollChangeActive AND "Unit1.EmNodes".slmRunning AND #emFeedback.isLinked);
   IF #_w8 AND "Unit1.Em5.ControlNodes".cmNgAndManualInputAxisY.monitoring.axisEnabled THEN
       "Unit1.Em5.ControlNodes".cmNgAndManualInputAxisY.commands.enableAxis := TRUE;
       "Unit1.Em5.HmiInterface".cmNgAndManualInputAxisY.commands.enableAxis := FALSE;
   END_IF;
   IF #_w8 AND "Unit1.Em5.ControlNodes".cmMagazineAxisZ.monitoring.axisEnabled THEN
       "Unit1.Em5.ControlNodes".cmMagazineAxisZ.commands.enableAxis := TRUE;
       "Unit1.Em5.HmiInterface".cmMagazineAxisZ.commands.enableAxis := FALSE;
   END_IF;
   #_w9 := NOT (NOT #statUnitStatus.mode.manual AND NOT #statUnitStatus.mode.maintenance) AND NOT "Unit1.EmNodes".allBrakeTest.monitoring.emStatus.busy[6] AND "Unit1.EmNodes".slmRunning;
   #_w10 := #_w9 AND NOT #statPulse[7];   // rising edge
   #statPulse[7] := #_w9;
   IF #_w10 AND "Unit1.Em5.ControlNodes".cmNgAndManualInputAxisY.monitoring.axisEnabled THEN
       "Unit1.Em5.HmiInterface".cmNgAndManualInputAxisY.commands.enableAxis := TRUE;
       "Unit1.Em5.ControlNodes".cmNgAndManualInputAxisY.commands.enableAxis := FALSE;
   END_IF;
   IF #_w10 AND "Unit1.Em5.ControlNodes".cmMagazineAxisZ.monitoring.axisEnabled THEN
       "Unit1.Em5.HmiInterface".cmMagazineAxisZ.commands.enableAxis := TRUE;
       "Unit1.Em5.ControlNodes".cmMagazineAxisZ.commands.enableAxis := FALSE;
   END_IF;
   #_w11 := NOT "Unit1.EmNodes".Zone1SafetyStatus.SFDoorOpen AND NOT "Unit1.EmNodes".SS1Extention AND "Unit1.EmNodes".slmRunning AND #emFeedback.isLinked AND NOT #statUnitStatus.mode.production;
   #_w12 := #_w11 AND NOT #statPulse[16];   // rising edge
   #statPulse[16] := #_w11;
   #_w13 := "Unit1.EmNodes".Zone1SafetyStatus.SFDoorOpen AND #statEnableManualCmds AND #emFeedback.isLinked AND NOT "Unit1.EmNodes".unitStatus.state.aborted;
   #_w14 := #_w13 AND NOT #statPulse[26];   // rising edge
   #statPulse[26] := #_w13;
   IF #_w12 OR #_w14 THEN
       "Unit1.Em5.HmiInterface".cmNgAndManualInputAxisY.commands.enableAxis := TRUE;
       "Unit1.Em5.ControlNodes".cmNgAndManualInputAxisY.commands.enableAxis := FALSE;
       "Unit1.Em5.HmiInterface".cmMagazineAxisZ.commands.enableAxis := TRUE;
       "Unit1.Em5.ControlNodes".cmMagazineAxisZ.commands.enableAxis := FALSE;
   END_IF;
   #statTonTimer[2].TON(IN := "Unit1.EmNodes".Zone1SafetyStatus.SFDoorOpen AND NOT "Unit1.EmNodes".LH_RollChangeActive AND NOT "Unit1.EmNodes".RH_RollChangeActive AND #emFeedback.isLinked,
                        PT := t#500ms);
   #_w15 := #statTonTimer[2].Q AND NOT #statPulse[17];   // rising edge
   #statPulse[17] := #statTonTimer[2].Q;
   #_w16 := NOT (NOT "Unit1.EmNodes".slmPowerOff AND NOT "Unit1.EmNodes".unitStatus.state.aborted AND NOT #statUnitStatus.mode.sleep AND NOT #statUnitStatus.mode.deepSleep) OR #_w15;
   IF #_w16 THEN
       "Unit1.Em5.HmiInterface".cmNgAndManualInputAxisY.commands.enableAxis := FALSE;
       "Unit1.Em5.HmiInterface".cmMagazineAxisZ.commands.enableAxis := FALSE;
   END_IF;
   IF #_w16 AND NOT "Unit1.EmNodes".allBrakeTest.monitoring.emStatus.busy[6] THEN
       "Unit1.Em5.ControlNodes".cmNgAndManualInputAxisY.commands.enableAxis := FALSE;
       "Unit1.Em5.ControlNodes".cmMagazineAxisZ.commands.enableAxis := FALSE;
   END_IF;
END_REGION

REGION Network 32: LBC_Axis64Pos Operation Mode
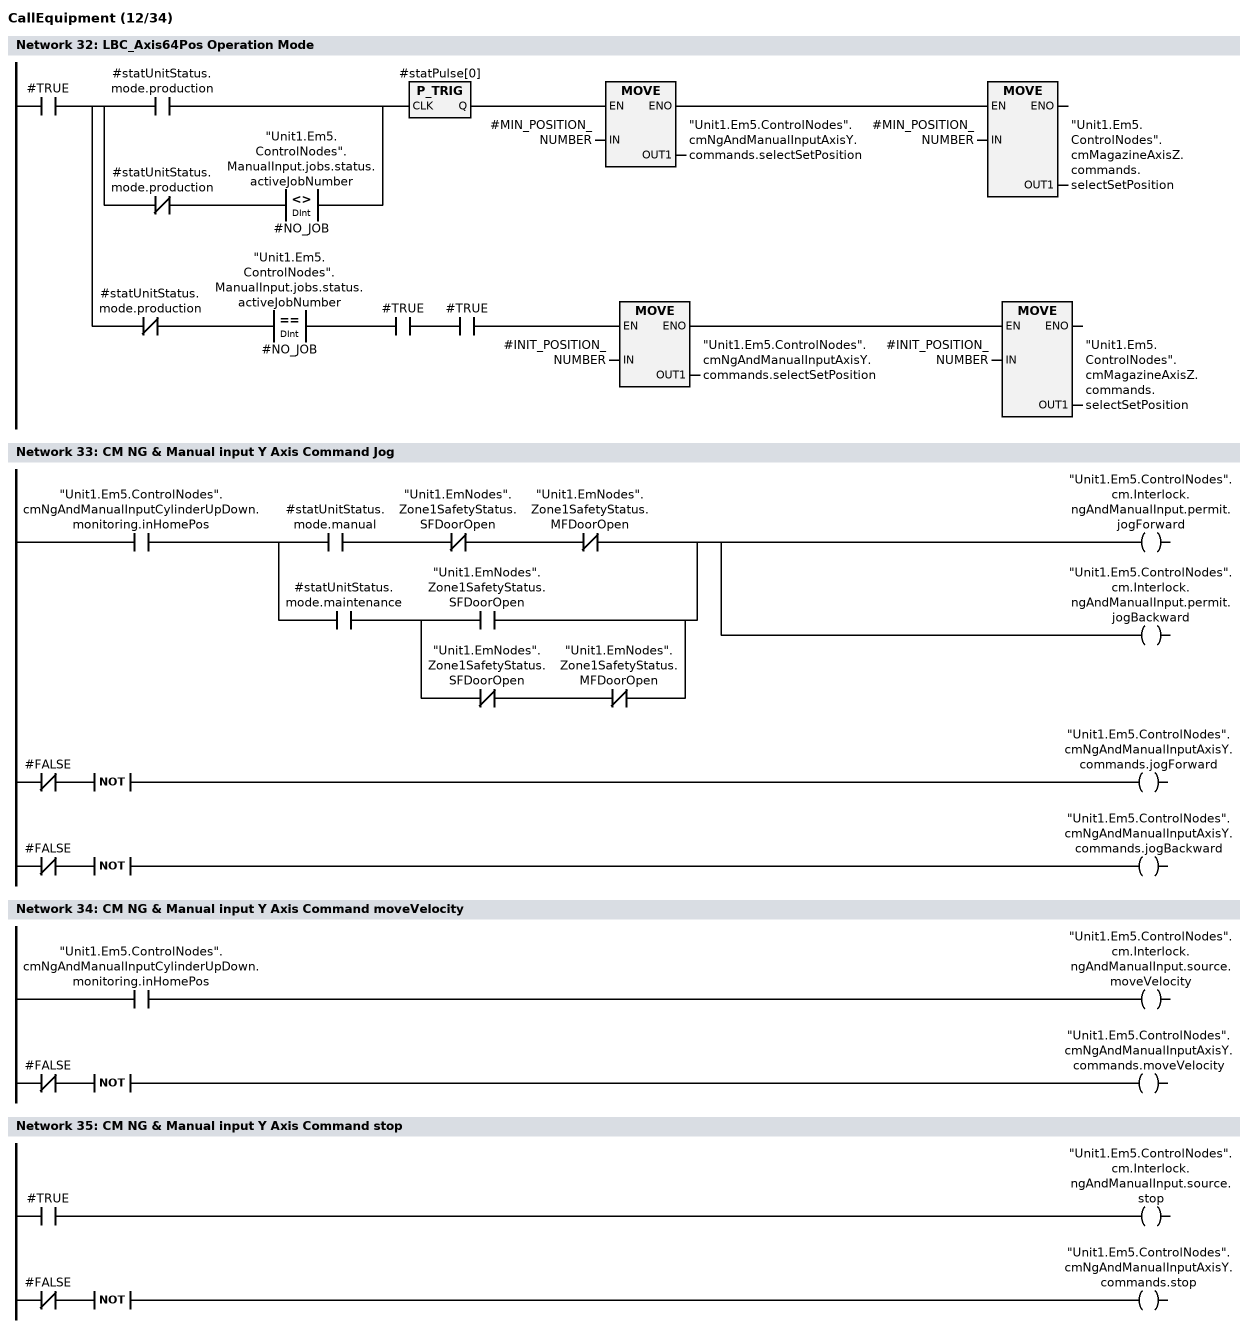
   RUNG wire#powerrail
      Contact( #TRUE )
      wire#w1
      Contact( #statUnitStatus.mode.production )
      wire#w2
      P_Trig( #statPulse[0] )
      Move(in := #MIN_POSITION_NUMBER, out1 => "Unit1.Em5.ControlNodes".cmNgAndManualInputAxisY.commands.selectSetPosition)
      Move(in := #MIN_POSITION_NUMBER, out1 => "Unit1.Em5.ControlNodes".cmMagazineAxisZ.commands.selectSetPosition)
   END_RUNG
   RUNG wire#w1
      I_Contact( #statUnitStatus.mode.production )
      { S7_Templates := "SrcType := DInt" } NE_Contact(in1 := "Unit1.Em5.ControlNodes".ManualInput.jobs.status.activeJobNumber, in2 := #NO_JOB)
   END_RUNG wire#w2
   RUNG wire#w1
      I_Contact( #statUnitStatus.mode.production )
      { S7_Templates := "SrcType := DInt" } EQ_Contact(in1 := "Unit1.Em5.ControlNodes".ManualInput.jobs.status.activeJobNumber, in2 := #NO_JOB)
      Contact( #TRUE )
      Contact( #TRUE )
      Move(in := #INIT_POSITION_NUMBER, out1 => "Unit1.Em5.ControlNodes".cmNgAndManualInputAxisY.commands.selectSetPosition)
      Move(in := #INIT_POSITION_NUMBER, out1 => "Unit1.Em5.ControlNodes".cmMagazineAxisZ.commands.selectSetPosition)
   END_RUNG
   // the same network as SCL:
   #_w1 := #TRUE AND (#statUnitStatus.mode.production OR (NOT #statUnitStatus.mode.production AND ("Unit1.Em5.ControlNodes".ManualInput.jobs.status.activeJobNumber <> #NO_JOB)));
   #_w2 := #_w1 AND NOT #statPulse[0];   // rising edge
   #statPulse[0] := #_w1;
   IF #_w2 THEN
       "Unit1.Em5.ControlNodes".cmNgAndManualInputAxisY.commands.selectSetPosition := #MIN_POSITION_NUMBER;
       "Unit1.Em5.ControlNodes".cmMagazineAxisZ.commands.selectSetPosition := #MIN_POSITION_NUMBER;
   END_IF;
   IF #TRUE AND NOT #statUnitStatus.mode.production AND ("Unit1.Em5.ControlNodes".ManualInput.jobs.status.activeJobNumber = #NO_JOB) AND #TRUE AND #TRUE THEN
       "Unit1.Em5.ControlNodes".cmNgAndManualInputAxisY.commands.selectSetPosition := #INIT_POSITION_NUMBER;
       "Unit1.Em5.ControlNodes".cmMagazineAxisZ.commands.selectSetPosition := #INIT_POSITION_NUMBER;
   END_IF;
END_REGION

REGION Network 33: CM NG & Manual input Y Axis Command Jog
   RUNG wire#powerrail
      Contact( "Unit1.Em5.ControlNodes".cmNgAndManualInputCylinderUpDown.monitoring.inHomePos )
      wire#w1
      Contact( #statUnitStatus.mode.manual )
      I_Contact( "Unit1.EmNodes".Zone1SafetyStatus.SFDoorOpen )
      I_Contact( "Unit1.EmNodes".Zone1SafetyStatus.MFDoorOpen )
      wire#w2
      Coil( "Unit1.Em5.ControlNodes".cm.Interlock.ngAndManualInput.permit.jogForward )
   END_RUNG
   RUNG wire#w1
      Contact( #statUnitStatus.mode.maintenance )
      wire#w3
      Contact( "Unit1.EmNodes".Zone1SafetyStatus.SFDoorOpen )
   END_RUNG wire#w2
   RUNG wire#w3
      I_Contact( "Unit1.EmNodes".Zone1SafetyStatus.SFDoorOpen )
      I_Contact( "Unit1.EmNodes".Zone1SafetyStatus.MFDoorOpen )
   END_RUNG wire#w2
   RUNG wire#w2
      Coil( "Unit1.Em5.ControlNodes".cm.Interlock.ngAndManualInput.permit.jogBackward )
   END_RUNG
   RUNG wire#powerrail
      I_Contact( #FALSE )
      Not()
      Coil( "Unit1.Em5.ControlNodes".cmNgAndManualInputAxisY.commands.jogForward )
   END_RUNG
   RUNG wire#powerrail
      I_Contact( #FALSE )
      Not()
      Coil( "Unit1.Em5.ControlNodes".cmNgAndManualInputAxisY.commands.jogBackward )
   END_RUNG
   // the same network as SCL:
   "Unit1.Em5.ControlNodes".cm.Interlock.ngAndManualInput.permit.jogForward := "Unit1.Em5.ControlNodes".cmNgAndManualInputCylinderUpDown.monitoring.inHomePos AND ((#statUnitStatus.mode.manual AND NOT "Unit1.EmNodes".Zone1SafetyStatus.SFDoorOpen AND NOT "Unit1.EmNodes".Zone1SafetyStatus.MFDoorOpen) OR (#statUnitStatus.mode.maintenance AND ("Unit1.EmNodes".Zone1SafetyStatus.SFDoorOpen OR (NOT "Unit1.EmNodes".Zone1SafetyStatus.SFDoorOpen AND NOT "Unit1.EmNodes".Zone1SafetyStatus.MFDoorOpen))));
   "Unit1.Em5.ControlNodes".cm.Interlock.ngAndManualInput.permit.jogBackward := "Unit1.Em5.ControlNodes".cm.Interlock.ngAndManualInput.permit.jogForward;
   "Unit1.Em5.ControlNodes".cmNgAndManualInputAxisY.commands.jogForward := NOT (NOT #FALSE);
   "Unit1.Em5.ControlNodes".cmNgAndManualInputAxisY.commands.jogBackward := NOT (NOT #FALSE);
END_REGION

REGION Network 34: CM NG & Manual input Y Axis Command moveVelocity
   RUNG wire#powerrail
      Contact( "Unit1.Em5.ControlNodes".cmNgAndManualInputCylinderUpDown.monitoring.inHomePos )
      Coil( "Unit1.Em5.ControlNodes".cm.Interlock.ngAndManualInput.source.moveVelocity )
   END_RUNG
   RUNG wire#powerrail
      I_Contact( #FALSE )
      Not()
      Coil( "Unit1.Em5.ControlNodes".cmNgAndManualInputAxisY.commands.moveVelocity )
   END_RUNG
   // the same network as SCL:
   "Unit1.Em5.ControlNodes".cm.Interlock.ngAndManualInput.source.moveVelocity := "Unit1.Em5.ControlNodes".cmNgAndManualInputCylinderUpDown.monitoring.inHomePos;
   "Unit1.Em5.ControlNodes".cmNgAndManualInputAxisY.commands.moveVelocity := NOT (NOT #FALSE);
END_REGION

REGION Network 35: CM NG & Manual input Y Axis Command stop
   RUNG wire#powerrail
      Contact( #TRUE )
      Coil( "Unit1.Em5.ControlNodes".cm.Interlock.ngAndManualInput.source.stop )
   END_RUNG
   RUNG wire#powerrail
      I_Contact( #FALSE )
      Not()
      Coil( "Unit1.Em5.ControlNodes".cmNgAndManualInputAxisY.commands.stop )
   END_RUNG
   // the same network as SCL:
   "Unit1.Em5.ControlNodes".cm.Interlock.ngAndManualInput.source.stop := #TRUE;
   "Unit1.Em5.ControlNodes".cmNgAndManualInputAxisY.commands.stop := NOT (NOT #FALSE);
END_REGION

REGION Network 36: CM NG & Manual input Y Axis Command fastStop
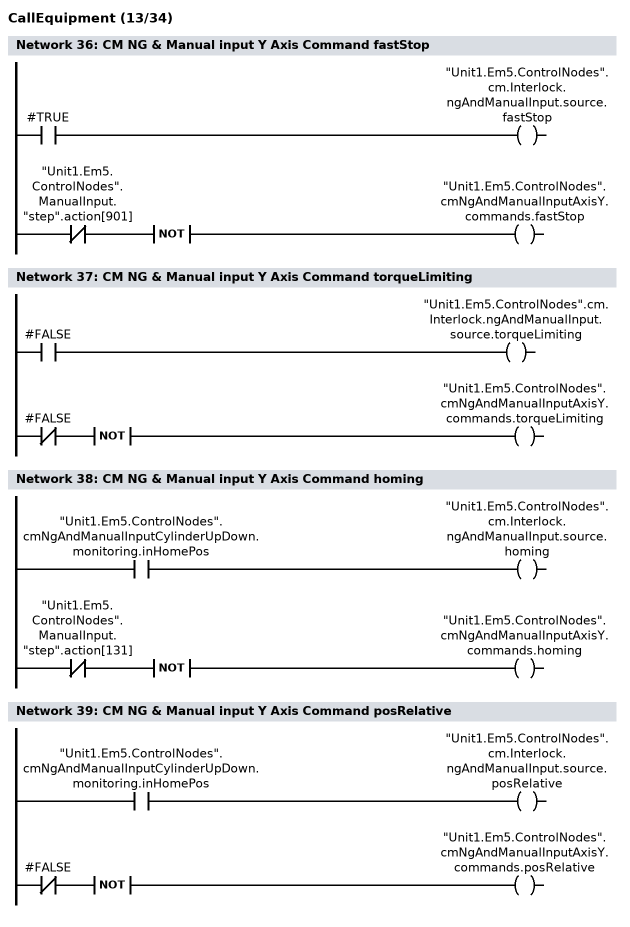
   RUNG wire#powerrail
      Contact( #TRUE )
      Coil( "Unit1.Em5.ControlNodes".cm.Interlock.ngAndManualInput.source.fastStop )
   END_RUNG
   RUNG wire#powerrail
      I_Contact( "Unit1.Em5.ControlNodes".ManualInput."step".action[901] )
      Not()
      Coil( "Unit1.Em5.ControlNodes".cmNgAndManualInputAxisY.commands.fastStop )
   END_RUNG
   // the same network as SCL:
   "Unit1.Em5.ControlNodes".cm.Interlock.ngAndManualInput.source.fastStop := #TRUE;
   "Unit1.Em5.ControlNodes".cmNgAndManualInputAxisY.commands.fastStop := NOT (NOT "Unit1.Em5.ControlNodes".ManualInput."step".action[901]);
END_REGION

REGION Network 37: CM NG & Manual input Y Axis Command torqueLimiting
   RUNG wire#powerrail
      Contact( #FALSE )
      Coil( "Unit1.Em5.ControlNodes".cm.Interlock.ngAndManualInput.source.torqueLimiting )
   END_RUNG
   RUNG wire#powerrail
      I_Contact( #FALSE )
      Not()
      Coil( "Unit1.Em5.ControlNodes".cmNgAndManualInputAxisY.commands.torqueLimiting )
   END_RUNG
   // the same network as SCL:
   "Unit1.Em5.ControlNodes".cm.Interlock.ngAndManualInput.source.torqueLimiting := #FALSE;
   "Unit1.Em5.ControlNodes".cmNgAndManualInputAxisY.commands.torqueLimiting := NOT (NOT #FALSE);
END_REGION

REGION Network 38: CM NG & Manual input Y Axis Command homing
   RUNG wire#powerrail
      Contact( "Unit1.Em5.ControlNodes".cmNgAndManualInputCylinderUpDown.monitoring.inHomePos )
      Coil( "Unit1.Em5.ControlNodes".cm.Interlock.ngAndManualInput.source.homing )
   END_RUNG
   RUNG wire#powerrail
      I_Contact( "Unit1.Em5.ControlNodes".ManualInput."step".action[131] )
      Not()
      Coil( "Unit1.Em5.ControlNodes".cmNgAndManualInputAxisY.commands.homing )
   END_RUNG
   // the same network as SCL:
   "Unit1.Em5.ControlNodes".cm.Interlock.ngAndManualInput.source.homing := "Unit1.Em5.ControlNodes".cmNgAndManualInputCylinderUpDown.monitoring.inHomePos;
   "Unit1.Em5.ControlNodes".cmNgAndManualInputAxisY.commands.homing := NOT (NOT "Unit1.Em5.ControlNodes".ManualInput."step".action[131]);
END_REGION

REGION Network 39: CM NG & Manual input Y Axis Command posRelative
   RUNG wire#powerrail
      Contact( "Unit1.Em5.ControlNodes".cmNgAndManualInputCylinderUpDown.monitoring.inHomePos )
      Coil( "Unit1.Em5.ControlNodes".cm.Interlock.ngAndManualInput.source.posRelative )
   END_RUNG
   RUNG wire#powerrail
      I_Contact( #FALSE )
      Not()
      Coil( "Unit1.Em5.ControlNodes".cmNgAndManualInputAxisY.commands.posRelative )
   END_RUNG
   // the same network as SCL:
   "Unit1.Em5.ControlNodes".cm.Interlock.ngAndManualInput.source.posRelative := "Unit1.Em5.ControlNodes".cmNgAndManualInputCylinderUpDown.monitoring.inHomePos;
   "Unit1.Em5.ControlNodes".cmNgAndManualInputAxisY.commands.posRelative := NOT (NOT #FALSE);
END_REGION

REGION Network 40: CM NG & Manual input Y Axis Command posAbsolute
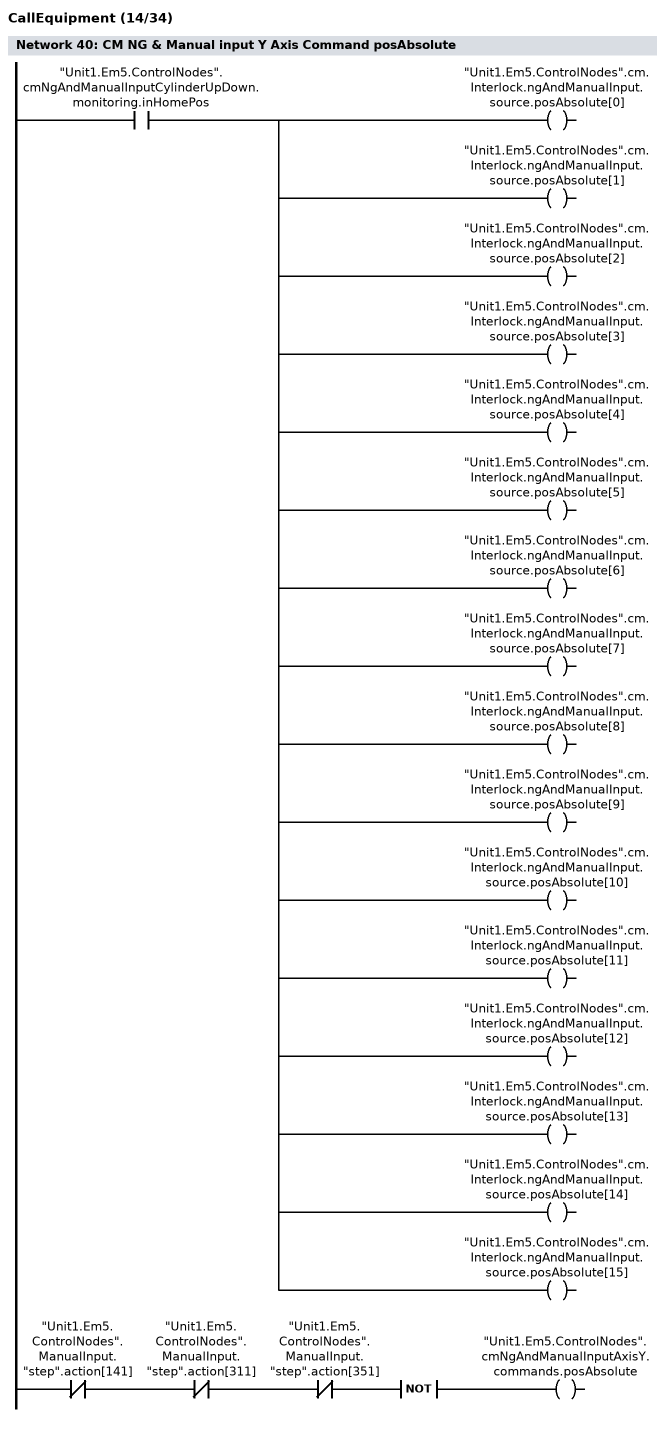
   RUNG wire#powerrail
      Contact( "Unit1.Em5.ControlNodes".cmNgAndManualInputCylinderUpDown.monitoring.inHomePos )
      wire#w1
      Coil( "Unit1.Em5.ControlNodes".cm.Interlock.ngAndManualInput.source.posAbsolute[0] )
   END_RUNG
   RUNG wire#w1
      Coil( "Unit1.Em5.ControlNodes".cm.Interlock.ngAndManualInput.source.posAbsolute[1] )
   END_RUNG
   RUNG wire#w1
      Coil( "Unit1.Em5.ControlNodes".cm.Interlock.ngAndManualInput.source.posAbsolute[2] )
   END_RUNG
   RUNG wire#w1
      Coil( "Unit1.Em5.ControlNodes".cm.Interlock.ngAndManualInput.source.posAbsolute[3] )
   END_RUNG
   RUNG wire#w1
      Coil( "Unit1.Em5.ControlNodes".cm.Interlock.ngAndManualInput.source.posAbsolute[4] )
   END_RUNG
   RUNG wire#w1
      Coil( "Unit1.Em5.ControlNodes".cm.Interlock.ngAndManualInput.source.posAbsolute[5] )
   END_RUNG
   RUNG wire#w1
      Coil( "Unit1.Em5.ControlNodes".cm.Interlock.ngAndManualInput.source.posAbsolute[6] )
   END_RUNG
   RUNG wire#w1
      Coil( "Unit1.Em5.ControlNodes".cm.Interlock.ngAndManualInput.source.posAbsolute[7] )
   END_RUNG
   RUNG wire#w1
      Coil( "Unit1.Em5.ControlNodes".cm.Interlock.ngAndManualInput.source.posAbsolute[8] )
   END_RUNG
   RUNG wire#w1
      Coil( "Unit1.Em5.ControlNodes".cm.Interlock.ngAndManualInput.source.posAbsolute[9] )
   END_RUNG
   RUNG wire#w1
      Coil( "Unit1.Em5.ControlNodes".cm.Interlock.ngAndManualInput.source.posAbsolute[10] )
   END_RUNG
   RUNG wire#w1
      Coil( "Unit1.Em5.ControlNodes".cm.Interlock.ngAndManualInput.source.posAbsolute[11] )
   END_RUNG
   RUNG wire#w1
      Coil( "Unit1.Em5.ControlNodes".cm.Interlock.ngAndManualInput.source.posAbsolute[12] )
   END_RUNG
   RUNG wire#w1
      Coil( "Unit1.Em5.ControlNodes".cm.Interlock.ngAndManualInput.source.posAbsolute[13] )
   END_RUNG
   RUNG wire#w1
      Coil( "Unit1.Em5.ControlNodes".cm.Interlock.ngAndManualInput.source.posAbsolute[14] )
   END_RUNG
   RUNG wire#w1
      Coil( "Unit1.Em5.ControlNodes".cm.Interlock.ngAndManualInput.source.posAbsolute[15] )
   END_RUNG
   RUNG wire#powerrail
      I_Contact( "Unit1.Em5.ControlNodes".ManualInput."step".action[141] )
      I_Contact( "Unit1.Em5.ControlNodes".ManualInput."step".action[311] )
      I_Contact( "Unit1.Em5.ControlNodes".ManualInput."step".action[351] )
      Not()
      Coil( "Unit1.Em5.ControlNodes".cmNgAndManualInputAxisY.commands.posAbsolute )
   END_RUNG
   // the same network as SCL:
   "Unit1.Em5.ControlNodes".cm.Interlock.ngAndManualInput.source.posAbsolute[0] := "Unit1.Em5.ControlNodes".cmNgAndManualInputCylinderUpDown.monitoring.inHomePos;
   "Unit1.Em5.ControlNodes".cm.Interlock.ngAndManualInput.source.posAbsolute[1] := "Unit1.Em5.ControlNodes".cmNgAndManualInputCylinderUpDown.monitoring.inHomePos;
   "Unit1.Em5.ControlNodes".cm.Interlock.ngAndManualInput.source.posAbsolute[2] := "Unit1.Em5.ControlNodes".cmNgAndManualInputCylinderUpDown.monitoring.inHomePos;
   "Unit1.Em5.ControlNodes".cm.Interlock.ngAndManualInput.source.posAbsolute[3] := "Unit1.Em5.ControlNodes".cmNgAndManualInputCylinderUpDown.monitoring.inHomePos;
   "Unit1.Em5.ControlNodes".cm.Interlock.ngAndManualInput.source.posAbsolute[4] := "Unit1.Em5.ControlNodes".cmNgAndManualInputCylinderUpDown.monitoring.inHomePos;
   "Unit1.Em5.ControlNodes".cm.Interlock.ngAndManualInput.source.posAbsolute[5] := "Unit1.Em5.ControlNodes".cmNgAndManualInputCylinderUpDown.monitoring.inHomePos;
   "Unit1.Em5.ControlNodes".cm.Interlock.ngAndManualInput.source.posAbsolute[6] := "Unit1.Em5.ControlNodes".cmNgAndManualInputCylinderUpDown.monitoring.inHomePos;
   "Unit1.Em5.ControlNodes".cm.Interlock.ngAndManualInput.source.posAbsolute[7] := "Unit1.Em5.ControlNodes".cmNgAndManualInputCylinderUpDown.monitoring.inHomePos;
   "Unit1.Em5.ControlNodes".cm.Interlock.ngAndManualInput.source.posAbsolute[8] := "Unit1.Em5.ControlNodes".cmNgAndManualInputCylinderUpDown.monitoring.inHomePos;
   "Unit1.Em5.ControlNodes".cm.Interlock.ngAndManualInput.source.posAbsolute[9] := "Unit1.Em5.ControlNodes".cmNgAndManualInputCylinderUpDown.monitoring.inHomePos;
   "Unit1.Em5.ControlNodes".cm.Interlock.ngAndManualInput.source.posAbsolute[10] := "Unit1.Em5.ControlNodes".cmNgAndManualInputCylinderUpDown.monitoring.inHomePos;
   "Unit1.Em5.ControlNodes".cm.Interlock.ngAndManualInput.source.posAbsolute[11] := "Unit1.Em5.ControlNodes".cmNgAndManualInputCylinderUpDown.monitoring.inHomePos;
   "Unit1.Em5.ControlNodes".cm.Interlock.ngAndManualInput.source.posAbsolute[12] := "Unit1.Em5.ControlNodes".cmNgAndManualInputCylinderUpDown.monitoring.inHomePos;
   "Unit1.Em5.ControlNodes".cm.Interlock.ngAndManualInput.source.posAbsolute[13] := "Unit1.Em5.ControlNodes".cmNgAndManualInputCylinderUpDown.monitoring.inHomePos;
   "Unit1.Em5.ControlNodes".cm.Interlock.ngAndManualInput.source.posAbsolute[14] := "Unit1.Em5.ControlNodes".cmNgAndManualInputCylinderUpDown.monitoring.inHomePos;
   "Unit1.Em5.ControlNodes".cm.Interlock.ngAndManualInput.source.posAbsolute[15] := "Unit1.Em5.ControlNodes".cmNgAndManualInputCylinderUpDown.monitoring.inHomePos;
   "Unit1.Em5.ControlNodes".cmNgAndManualInputAxisY.commands.posAbsolute := NOT (NOT "Unit1.Em5.ControlNodes".ManualInput."step".action[141] AND NOT "Unit1.Em5.ControlNodes".ManualInput."step".action[311] AND NOT "Unit1.Em5.ControlNodes".ManualInput."step".action[351]);
END_REGION

REGION Network 41: Call CM NG & Manual input Y Axis (LER_Interlock Summary)
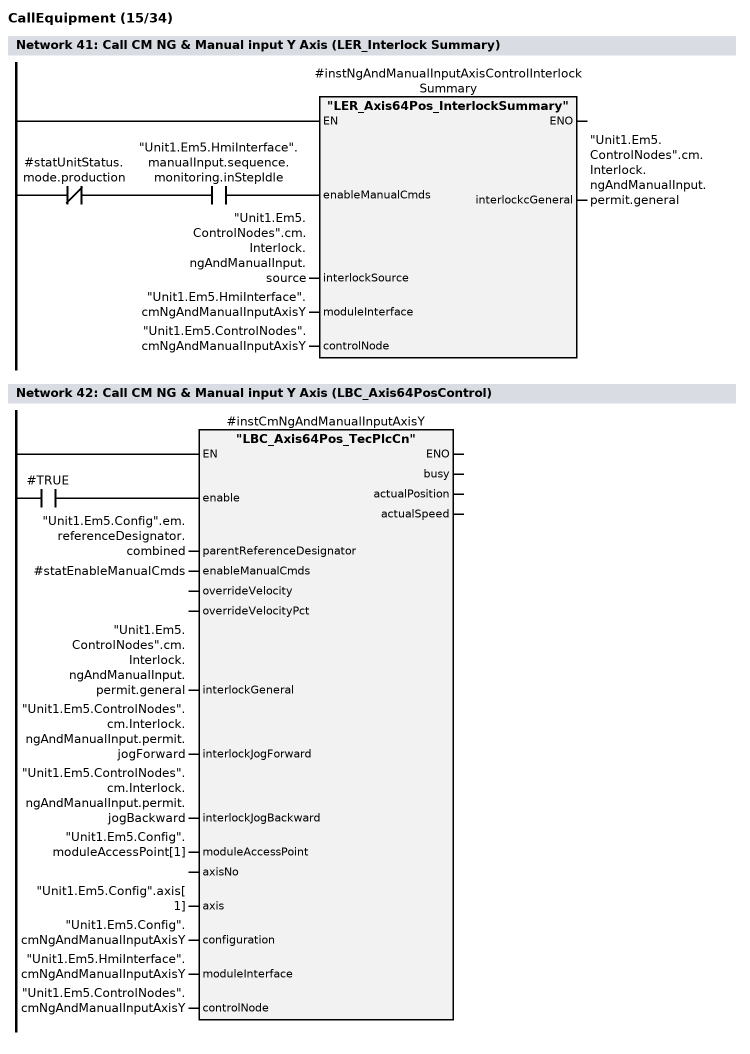
   RUNG wire#powerrail
      #instNgAndManualInputAxisControlInterlockSummary(enableManualCmds := wire#w1, interlockSource := "Unit1.Em5.ControlNodes".cm.Interlock.ngAndManualInput.source, moduleInterface := "Unit1.Em5.HmiInterface".cmNgAndManualInputAxisY, controlNode := "Unit1.Em5.ControlNodes".cmNgAndManualInputAxisY, interlockcGeneral => "Unit1.Em5.ControlNodes".cm.Interlock.ngAndManualInput.permit.general)
   END_RUNG
   RUNG wire#powerrail
      I_Contact( #statUnitStatus.mode.production )
      Contact( "Unit1.Em5.HmiInterface".manualInput.sequence.monitoring.inStepIdle )
   END_RUNG wire#w1
   // the same network as SCL:
   #instNgAndManualInputAxisControlInterlockSummary(enableManualCmds := NOT #statUnitStatus.mode.production AND "Unit1.Em5.HmiInterface".manualInput.sequence.monitoring.inStepIdle,   // "LER_Axis64Pos_InterlockSummary"
                           interlockSource := "Unit1.Em5.ControlNodes".cm.Interlock.ngAndManualInput.source,
                           moduleInterface := "Unit1.Em5.HmiInterface".cmNgAndManualInputAxisY,
                           controlNode := "Unit1.Em5.ControlNodes".cmNgAndManualInputAxisY,
                           interlockcGeneral => "Unit1.Em5.ControlNodes".cm.Interlock.ngAndManualInput.permit.general);
END_REGION

REGION Network 42: Call CM NG & Manual input Y Axis (LBC_Axis64PosControl)
   RUNG wire#powerrail
      #instCmNgAndManualInputAxisY(enable := wire#w1, parentReferenceDesignator := "Unit1.Em5.Config".em.referenceDesignator.combined, enableManualCmds := #statEnableManualCmds, overrideVelocity :=, overrideVelocityPct :=, interlockGeneral := "Unit1.Em5.ControlNodes".cm.Interlock.ngAndManualInput.permit.general, interlockJogForward := "Unit1.Em5.ControlNodes".cm.Interlock.ngAndManualInput.permit.jogForward, interlockJogBackward := "Unit1.Em5.ControlNodes".cm.Interlock.ngAndManualInput.permit.jogBackward, moduleAccessPoint := "Unit1.Em5.Config".moduleAccessPoint[1], axisNo :=, axis := "Unit1.Em5.Config".axis[1], configuration := "Unit1.Em5.Config".cmNgAndManualInputAxisY, moduleInterface := "Unit1.Em5.HmiInterface".cmNgAndManualInputAxisY, controlNode := "Unit1.Em5.ControlNodes".cmNgAndManualInputAxisY, busy =>, actualPosition =>, actualSpeed =>)
   END_RUNG
   RUNG wire#powerrail
      Contact( #TRUE )
   END_RUNG wire#w1
   // the same network as SCL:
   #instCmNgAndManualInputAxisY(enable := #TRUE,   // "LBC_Axis64Pos_TecPlcCn"
                           parentReferenceDesignator := "Unit1.Em5.Config".em.referenceDesignator.combined,
                           enableManualCmds := #statEnableManualCmds,
                           interlockGeneral := "Unit1.Em5.ControlNodes".cm.Interlock.ngAndManualInput.permit.general,
                           interlockJogForward := "Unit1.Em5.ControlNodes".cm.Interlock.ngAndManualInput.permit.jogForward,
                           interlockJogBackward := "Unit1.Em5.ControlNodes".cm.Interlock.ngAndManualInput.permit.jogBackward,
                           moduleAccessPoint := "Unit1.Em5.Config".moduleAccessPoint[1],
                           axis := "Unit1.Em5.Config".axis[1],
                           configuration := "Unit1.Em5.Config".cmNgAndManualInputAxisY,
                           moduleInterface := "Unit1.Em5.HmiInterface".cmNgAndManualInputAxisY,
                           controlNode := "Unit1.Em5.ControlNodes".cmNgAndManualInputAxisY);
END_REGION

REGION Network 43: Call CM NG & Manual input Y Axis (LER_ServoTorqueCal)
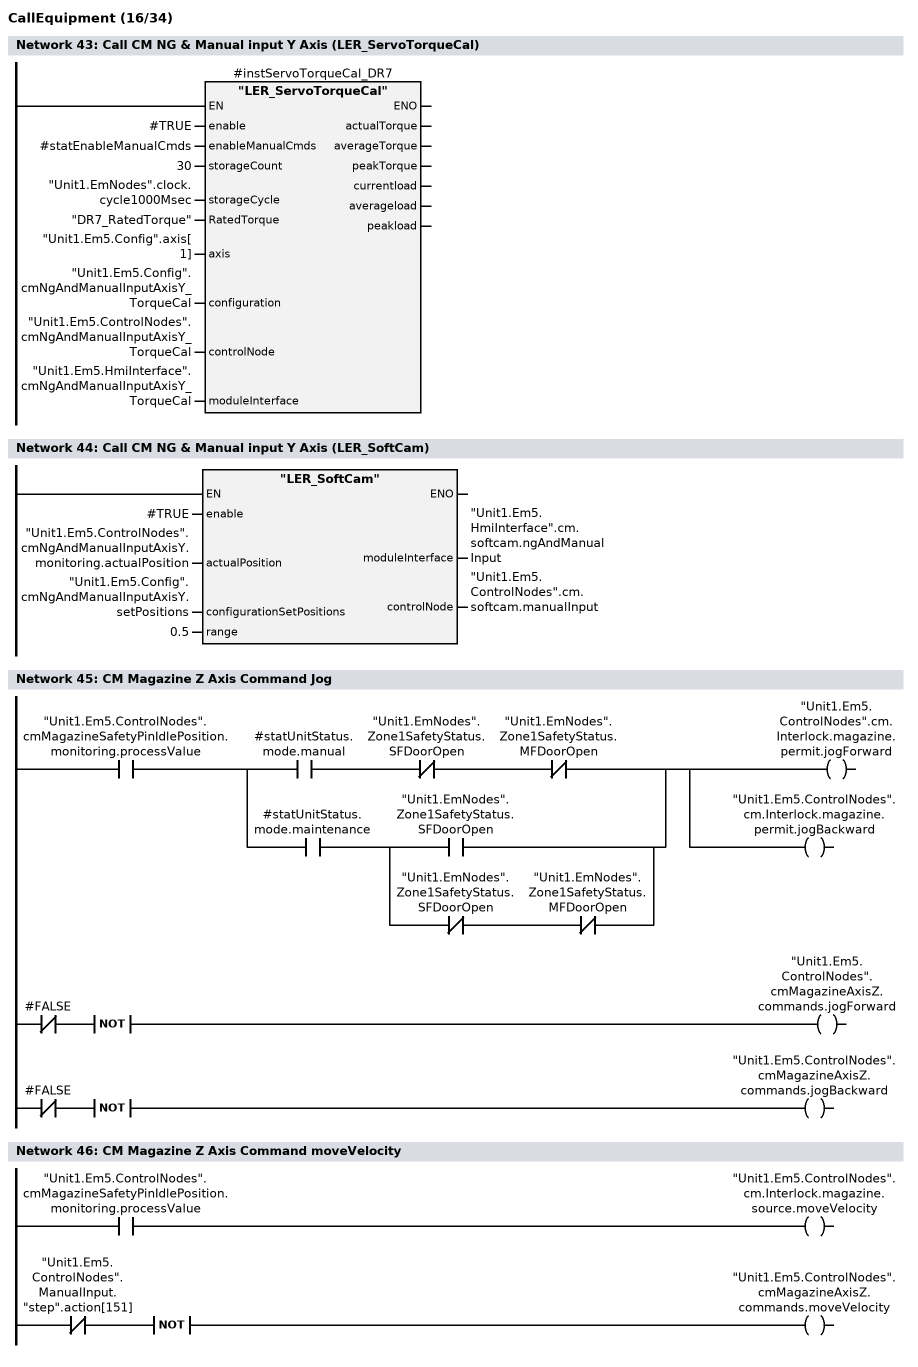
   RUNG wire#powerrail
      #instServoTorqueCal_DR7(enable := #TRUE, enableManualCmds := #statEnableManualCmds, storageCount := 30, storageCycle := "Unit1.EmNodes".clock.cycle1000Msec, RatedTorque := "DR7_RatedTorque", axis := "Unit1.Em5.Config".axis[1], configuration := "Unit1.Em5.Config".cmNgAndManualInputAxisY_TorqueCal, controlNode := "Unit1.Em5.ControlNodes".cmNgAndManualInputAxisY_TorqueCal, moduleInterface := "Unit1.Em5.HmiInterface".cmNgAndManualInputAxisY_TorqueCal, actualTorque =>, averageTorque =>, peakTorque =>, currentload =>, averageload =>, peakload =>)
   END_RUNG
   // the same network as SCL:
   #instServoTorqueCal_DR7(enable := #TRUE,   // "LER_ServoTorqueCal"
                           enableManualCmds := #statEnableManualCmds,
                           storageCount := 30,
                           storageCycle := "Unit1.EmNodes".clock.cycle1000Msec,
                           RatedTorque := "DR7_RatedTorque",
                           axis := "Unit1.Em5.Config".axis[1],
                           configuration := "Unit1.Em5.Config".cmNgAndManualInputAxisY_TorqueCal,
                           controlNode := "Unit1.Em5.ControlNodes".cmNgAndManualInputAxisY_TorqueCal,
                           moduleInterface := "Unit1.Em5.HmiInterface".cmNgAndManualInputAxisY_TorqueCal);
END_REGION

REGION Network 44: Call CM NG & Manual input Y Axis (LER_SoftCam)
   RUNG wire#powerrail
      "LER_SoftCam"(enable := #TRUE, actualPosition := "Unit1.Em5.ControlNodes".cmNgAndManualInputAxisY.monitoring.actualPosition, configurationSetPositions := "Unit1.Em5.Config".cmNgAndManualInputAxisY.setPositions, range := 0.5, moduleInterface => "Unit1.Em5.HmiInterface".cm.softcam.ngAndManualInput, controlNode => "Unit1.Em5.ControlNodes".cm.softcam.manualInput)
   END_RUNG
   // the same network as SCL:
   "LER_SoftCam"(enable := #TRUE,
                 actualPosition := "Unit1.Em5.ControlNodes".cmNgAndManualInputAxisY.monitoring.actualPosition,
                 configurationSetPositions := "Unit1.Em5.Config".cmNgAndManualInputAxisY.setPositions,
                 range := 0.5,
                 moduleInterface => "Unit1.Em5.HmiInterface".cm.softcam.ngAndManualInput,
                 controlNode => "Unit1.Em5.ControlNodes".cm.softcam.manualInput);
END_REGION

REGION Network 45: CM Magazine Z Axis Command Jog
   RUNG wire#powerrail
      Contact( "Unit1.Em5.ControlNodes".cmMagazineSafetyPinIdlePosition.monitoring.processValue )
      wire#w1
      Contact( #statUnitStatus.mode.manual )
      I_Contact( "Unit1.EmNodes".Zone1SafetyStatus.SFDoorOpen )
      I_Contact( "Unit1.EmNodes".Zone1SafetyStatus.MFDoorOpen )
      wire#w2
      Coil( "Unit1.Em5.ControlNodes".cm.Interlock.magazine.permit.jogForward )
   END_RUNG
   RUNG wire#w1
      Contact( #statUnitStatus.mode.maintenance )
      wire#w3
      Contact( "Unit1.EmNodes".Zone1SafetyStatus.SFDoorOpen )
   END_RUNG wire#w2
   RUNG wire#w3
      I_Contact( "Unit1.EmNodes".Zone1SafetyStatus.SFDoorOpen )
      I_Contact( "Unit1.EmNodes".Zone1SafetyStatus.MFDoorOpen )
   END_RUNG wire#w2
   RUNG wire#w2
      Coil( "Unit1.Em5.ControlNodes".cm.Interlock.magazine.permit.jogBackward )
   END_RUNG
   RUNG wire#powerrail
      I_Contact( #FALSE )
      Not()
      Coil( "Unit1.Em5.ControlNodes".cmMagazineAxisZ.commands.jogForward )
   END_RUNG
   RUNG wire#powerrail
      I_Contact( #FALSE )
      Not()
      Coil( "Unit1.Em5.ControlNodes".cmMagazineAxisZ.commands.jogBackward )
   END_RUNG
   // the same network as SCL:
   "Unit1.Em5.ControlNodes".cm.Interlock.magazine.permit.jogForward := "Unit1.Em5.ControlNodes".cmMagazineSafetyPinIdlePosition.monitoring.processValue AND ((#statUnitStatus.mode.manual AND NOT "Unit1.EmNodes".Zone1SafetyStatus.SFDoorOpen AND NOT "Unit1.EmNodes".Zone1SafetyStatus.MFDoorOpen) OR (#statUnitStatus.mode.maintenance AND ("Unit1.EmNodes".Zone1SafetyStatus.SFDoorOpen OR (NOT "Unit1.EmNodes".Zone1SafetyStatus.SFDoorOpen AND NOT "Unit1.EmNodes".Zone1SafetyStatus.MFDoorOpen))));
   "Unit1.Em5.ControlNodes".cm.Interlock.magazine.permit.jogBackward := "Unit1.Em5.ControlNodes".cm.Interlock.magazine.permit.jogForward;
   "Unit1.Em5.ControlNodes".cmMagazineAxisZ.commands.jogForward := NOT (NOT #FALSE);
   "Unit1.Em5.ControlNodes".cmMagazineAxisZ.commands.jogBackward := NOT (NOT #FALSE);
END_REGION

REGION Network 46: CM Magazine Z Axis Command moveVelocity
   RUNG wire#powerrail
      Contact( "Unit1.Em5.ControlNodes".cmMagazineSafetyPinIdlePosition.monitoring.processValue )
      Coil( "Unit1.Em5.ControlNodes".cm.Interlock.magazine.source.moveVelocity )
   END_RUNG
   RUNG wire#powerrail
      I_Contact( "Unit1.Em5.ControlNodes".ManualInput."step".action[151] )
      Not()
      Coil( "Unit1.Em5.ControlNodes".cmMagazineAxisZ.commands.moveVelocity )
   END_RUNG
   // the same network as SCL:
   "Unit1.Em5.ControlNodes".cm.Interlock.magazine.source.moveVelocity := "Unit1.Em5.ControlNodes".cmMagazineSafetyPinIdlePosition.monitoring.processValue;
   "Unit1.Em5.ControlNodes".cmMagazineAxisZ.commands.moveVelocity := NOT (NOT "Unit1.Em5.ControlNodes".ManualInput."step".action[151]);
END_REGION

REGION Network 47: CM Magazine Z Axis Command stop
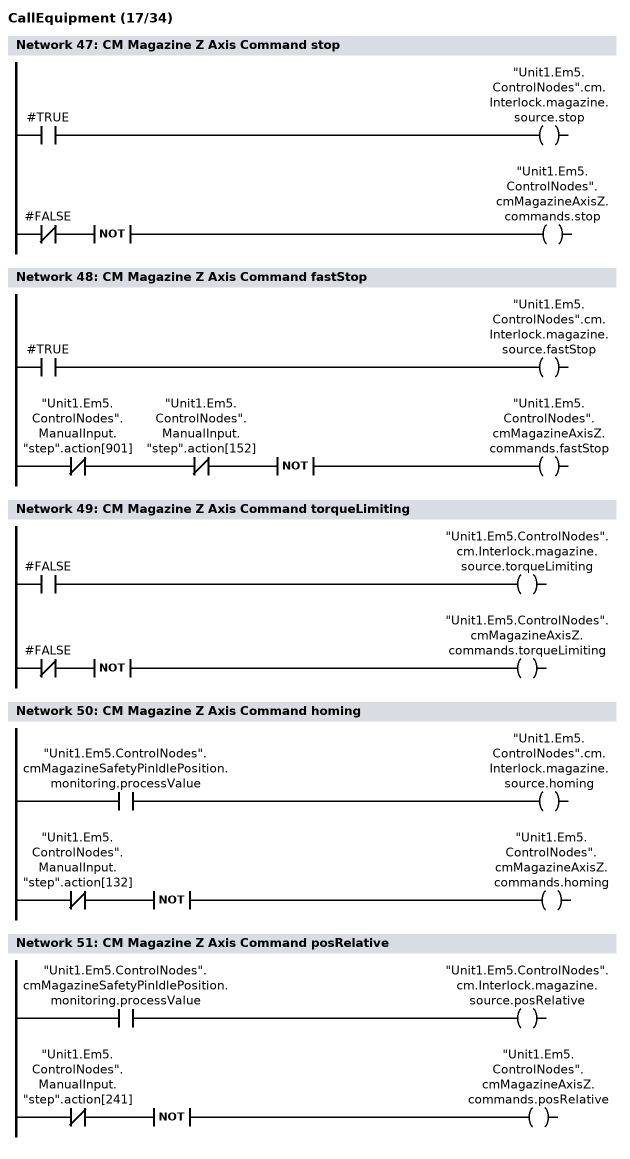
   RUNG wire#powerrail
      Contact( #TRUE )
      Coil( "Unit1.Em5.ControlNodes".cm.Interlock.magazine.source.stop )
   END_RUNG
   RUNG wire#powerrail
      I_Contact( #FALSE )
      Not()
      Coil( "Unit1.Em5.ControlNodes".cmMagazineAxisZ.commands.stop )
   END_RUNG
   // the same network as SCL:
   "Unit1.Em5.ControlNodes".cm.Interlock.magazine.source.stop := #TRUE;
   "Unit1.Em5.ControlNodes".cmMagazineAxisZ.commands.stop := NOT (NOT #FALSE);
END_REGION

REGION Network 48: CM Magazine Z Axis Command fastStop
   RUNG wire#powerrail
      Contact( #TRUE )
      Coil( "Unit1.Em5.ControlNodes".cm.Interlock.magazine.source.fastStop )
   END_RUNG
   RUNG wire#powerrail
      I_Contact( "Unit1.Em5.ControlNodes".ManualInput."step".action[901] )
      I_Contact( "Unit1.Em5.ControlNodes".ManualInput."step".action[152] )
      Not()
      Coil( "Unit1.Em5.ControlNodes".cmMagazineAxisZ.commands.fastStop )
   END_RUNG
   // the same network as SCL:
   "Unit1.Em5.ControlNodes".cm.Interlock.magazine.source.fastStop := #TRUE;
   "Unit1.Em5.ControlNodes".cmMagazineAxisZ.commands.fastStop := NOT (NOT "Unit1.Em5.ControlNodes".ManualInput."step".action[901] AND NOT "Unit1.Em5.ControlNodes".ManualInput."step".action[152]);
END_REGION

REGION Network 49: CM Magazine Z Axis Command torqueLimiting
   RUNG wire#powerrail
      Contact( #FALSE )
      Coil( "Unit1.Em5.ControlNodes".cm.Interlock.magazine.source.torqueLimiting )
   END_RUNG
   RUNG wire#powerrail
      I_Contact( #FALSE )
      Not()
      Coil( "Unit1.Em5.ControlNodes".cmMagazineAxisZ.commands.torqueLimiting )
   END_RUNG
   // the same network as SCL:
   "Unit1.Em5.ControlNodes".cm.Interlock.magazine.source.torqueLimiting := #FALSE;
   "Unit1.Em5.ControlNodes".cmMagazineAxisZ.commands.torqueLimiting := NOT (NOT #FALSE);
END_REGION

REGION Network 50: CM Magazine Z Axis Command homing
   RUNG wire#powerrail
      Contact( "Unit1.Em5.ControlNodes".cmMagazineSafetyPinIdlePosition.monitoring.processValue )
      Coil( "Unit1.Em5.ControlNodes".cm.Interlock.magazine.source.homing )
   END_RUNG
   RUNG wire#powerrail
      I_Contact( "Unit1.Em5.ControlNodes".ManualInput."step".action[132] )
      Not()
      Coil( "Unit1.Em5.ControlNodes".cmMagazineAxisZ.commands.homing )
   END_RUNG
   // the same network as SCL:
   "Unit1.Em5.ControlNodes".cm.Interlock.magazine.source.homing := "Unit1.Em5.ControlNodes".cmMagazineSafetyPinIdlePosition.monitoring.processValue;
   "Unit1.Em5.ControlNodes".cmMagazineAxisZ.commands.homing := NOT (NOT "Unit1.Em5.ControlNodes".ManualInput."step".action[132]);
END_REGION

REGION Network 51: CM Magazine Z Axis Command posRelative
   RUNG wire#powerrail
      Contact( "Unit1.Em5.ControlNodes".cmMagazineSafetyPinIdlePosition.monitoring.processValue )
      Coil( "Unit1.Em5.ControlNodes".cm.Interlock.magazine.source.posRelative )
   END_RUNG
   RUNG wire#powerrail
      I_Contact( "Unit1.Em5.ControlNodes".ManualInput."step".action[241] )
      Not()
      Coil( "Unit1.Em5.ControlNodes".cmMagazineAxisZ.commands.posRelative )
   END_RUNG
   // the same network as SCL:
   "Unit1.Em5.ControlNodes".cm.Interlock.magazine.source.posRelative := "Unit1.Em5.ControlNodes".cmMagazineSafetyPinIdlePosition.monitoring.processValue;
   "Unit1.Em5.ControlNodes".cmMagazineAxisZ.commands.posRelative := NOT (NOT "Unit1.Em5.ControlNodes".ManualInput."step".action[241]);
END_REGION

REGION Network 52: CM Magazine Z Axis Command posAbsolute
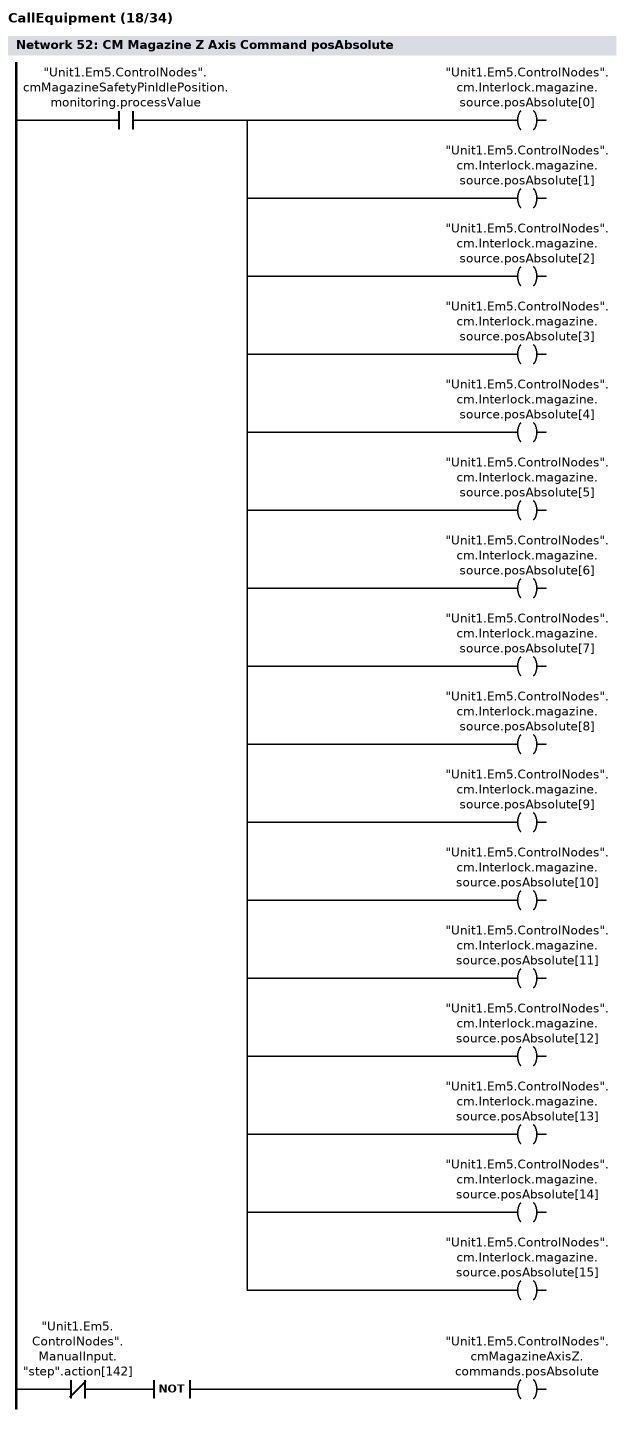
   RUNG wire#powerrail
      Contact( "Unit1.Em5.ControlNodes".cmMagazineSafetyPinIdlePosition.monitoring.processValue )
      wire#w1
      Coil( "Unit1.Em5.ControlNodes".cm.Interlock.magazine.source.posAbsolute[0] )
   END_RUNG
   RUNG wire#w1
      Coil( "Unit1.Em5.ControlNodes".cm.Interlock.magazine.source.posAbsolute[1] )
   END_RUNG
   RUNG wire#w1
      Coil( "Unit1.Em5.ControlNodes".cm.Interlock.magazine.source.posAbsolute[2] )
   END_RUNG
   RUNG wire#w1
      Coil( "Unit1.Em5.ControlNodes".cm.Interlock.magazine.source.posAbsolute[3] )
   END_RUNG
   RUNG wire#w1
      Coil( "Unit1.Em5.ControlNodes".cm.Interlock.magazine.source.posAbsolute[4] )
   END_RUNG
   RUNG wire#w1
      Coil( "Unit1.Em5.ControlNodes".cm.Interlock.magazine.source.posAbsolute[5] )
   END_RUNG
   RUNG wire#w1
      Coil( "Unit1.Em5.ControlNodes".cm.Interlock.magazine.source.posAbsolute[6] )
   END_RUNG
   RUNG wire#w1
      Coil( "Unit1.Em5.ControlNodes".cm.Interlock.magazine.source.posAbsolute[7] )
   END_RUNG
   RUNG wire#w1
      Coil( "Unit1.Em5.ControlNodes".cm.Interlock.magazine.source.posAbsolute[8] )
   END_RUNG
   RUNG wire#w1
      Coil( "Unit1.Em5.ControlNodes".cm.Interlock.magazine.source.posAbsolute[9] )
   END_RUNG
   RUNG wire#w1
      Coil( "Unit1.Em5.ControlNodes".cm.Interlock.magazine.source.posAbsolute[10] )
   END_RUNG
   RUNG wire#w1
      Coil( "Unit1.Em5.ControlNodes".cm.Interlock.magazine.source.posAbsolute[11] )
   END_RUNG
   RUNG wire#w1
      Coil( "Unit1.Em5.ControlNodes".cm.Interlock.magazine.source.posAbsolute[12] )
   END_RUNG
   RUNG wire#w1
      Coil( "Unit1.Em5.ControlNodes".cm.Interlock.magazine.source.posAbsolute[13] )
   END_RUNG
   RUNG wire#w1
      Coil( "Unit1.Em5.ControlNodes".cm.Interlock.magazine.source.posAbsolute[14] )
   END_RUNG
   RUNG wire#w1
      Coil( "Unit1.Em5.ControlNodes".cm.Interlock.magazine.source.posAbsolute[15] )
   END_RUNG
   RUNG wire#powerrail
      I_Contact( "Unit1.Em5.ControlNodes".ManualInput."step".action[142] )
      Not()
      Coil( "Unit1.Em5.ControlNodes".cmMagazineAxisZ.commands.posAbsolute )
   END_RUNG
   // the same network as SCL:
   "Unit1.Em5.ControlNodes".cm.Interlock.magazine.source.posAbsolute[0] := "Unit1.Em5.ControlNodes".cmMagazineSafetyPinIdlePosition.monitoring.processValue;
   "Unit1.Em5.ControlNodes".cm.Interlock.magazine.source.posAbsolute[1] := "Unit1.Em5.ControlNodes".cmMagazineSafetyPinIdlePosition.monitoring.processValue;
   "Unit1.Em5.ControlNodes".cm.Interlock.magazine.source.posAbsolute[2] := "Unit1.Em5.ControlNodes".cmMagazineSafetyPinIdlePosition.monitoring.processValue;
   "Unit1.Em5.ControlNodes".cm.Interlock.magazine.source.posAbsolute[3] := "Unit1.Em5.ControlNodes".cmMagazineSafetyPinIdlePosition.monitoring.processValue;
   "Unit1.Em5.ControlNodes".cm.Interlock.magazine.source.posAbsolute[4] := "Unit1.Em5.ControlNodes".cmMagazineSafetyPinIdlePosition.monitoring.processValue;
   "Unit1.Em5.ControlNodes".cm.Interlock.magazine.source.posAbsolute[5] := "Unit1.Em5.ControlNodes".cmMagazineSafetyPinIdlePosition.monitoring.processValue;
   "Unit1.Em5.ControlNodes".cm.Interlock.magazine.source.posAbsolute[6] := "Unit1.Em5.ControlNodes".cmMagazineSafetyPinIdlePosition.monitoring.processValue;
   "Unit1.Em5.ControlNodes".cm.Interlock.magazine.source.posAbsolute[7] := "Unit1.Em5.ControlNodes".cmMagazineSafetyPinIdlePosition.monitoring.processValue;
   "Unit1.Em5.ControlNodes".cm.Interlock.magazine.source.posAbsolute[8] := "Unit1.Em5.ControlNodes".cmMagazineSafetyPinIdlePosition.monitoring.processValue;
   "Unit1.Em5.ControlNodes".cm.Interlock.magazine.source.posAbsolute[9] := "Unit1.Em5.ControlNodes".cmMagazineSafetyPinIdlePosition.monitoring.processValue;
   "Unit1.Em5.ControlNodes".cm.Interlock.magazine.source.posAbsolute[10] := "Unit1.Em5.ControlNodes".cmMagazineSafetyPinIdlePosition.monitoring.processValue;
   "Unit1.Em5.ControlNodes".cm.Interlock.magazine.source.posAbsolute[11] := "Unit1.Em5.ControlNodes".cmMagazineSafetyPinIdlePosition.monitoring.processValue;
   "Unit1.Em5.ControlNodes".cm.Interlock.magazine.source.posAbsolute[12] := "Unit1.Em5.ControlNodes".cmMagazineSafetyPinIdlePosition.monitoring.processValue;
   "Unit1.Em5.ControlNodes".cm.Interlock.magazine.source.posAbsolute[13] := "Unit1.Em5.ControlNodes".cmMagazineSafetyPinIdlePosition.monitoring.processValue;
   "Unit1.Em5.ControlNodes".cm.Interlock.magazine.source.posAbsolute[14] := "Unit1.Em5.ControlNodes".cmMagazineSafetyPinIdlePosition.monitoring.processValue;
   "Unit1.Em5.ControlNodes".cm.Interlock.magazine.source.posAbsolute[15] := "Unit1.Em5.ControlNodes".cmMagazineSafetyPinIdlePosition.monitoring.processValue;
   "Unit1.Em5.ControlNodes".cmMagazineAxisZ.commands.posAbsolute := NOT (NOT "Unit1.Em5.ControlNodes".ManualInput."step".action[142]);
END_REGION

REGION Network 53: Call CM Magazine Z Axis (LER_Interlock Summary)
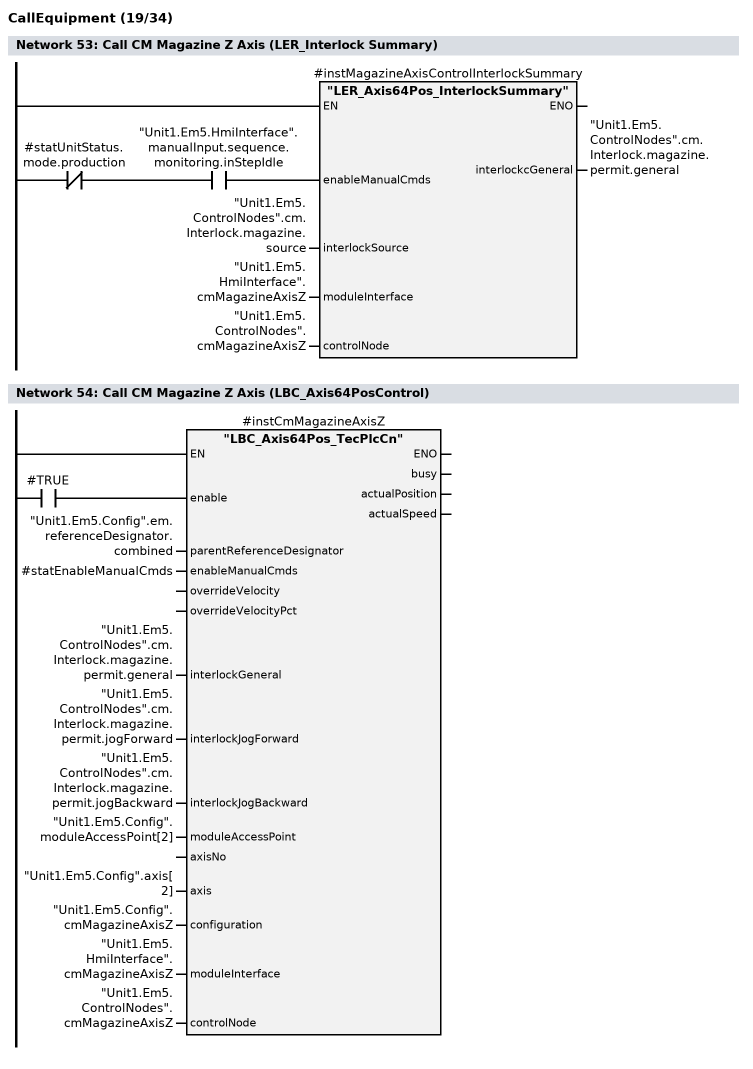
   RUNG wire#powerrail
      #instMagazineAxisControlInterlockSummary(enableManualCmds := wire#w1, interlockSource := "Unit1.Em5.ControlNodes".cm.Interlock.magazine.source, moduleInterface := "Unit1.Em5.HmiInterface".cmMagazineAxisZ, controlNode := "Unit1.Em5.ControlNodes".cmMagazineAxisZ, interlockcGeneral => "Unit1.Em5.ControlNodes".cm.Interlock.magazine.permit.general)
   END_RUNG
   RUNG wire#powerrail
      I_Contact( #statUnitStatus.mode.production )
      Contact( "Unit1.Em5.HmiInterface".manualInput.sequence.monitoring.inStepIdle )
   END_RUNG wire#w1
   // the same network as SCL:
   #instMagazineAxisControlInterlockSummary(enableManualCmds := NOT #statUnitStatus.mode.production AND "Unit1.Em5.HmiInterface".manualInput.sequence.monitoring.inStepIdle,   // "LER_Axis64Pos_InterlockSummary"
                           interlockSource := "Unit1.Em5.ControlNodes".cm.Interlock.magazine.source,
                           moduleInterface := "Unit1.Em5.HmiInterface".cmMagazineAxisZ,
                           controlNode := "Unit1.Em5.ControlNodes".cmMagazineAxisZ,
                           interlockcGeneral => "Unit1.Em5.ControlNodes".cm.Interlock.magazine.permit.general);
END_REGION

REGION Network 54: Call CM Magazine Z Axis (LBC_Axis64PosControl)
   RUNG wire#powerrail
      #instCmMagazineAxisZ(enable := wire#w1, parentReferenceDesignator := "Unit1.Em5.Config".em.referenceDesignator.combined, enableManualCmds := #statEnableManualCmds, overrideVelocity :=, overrideVelocityPct :=, interlockGeneral := "Unit1.Em5.ControlNodes".cm.Interlock.magazine.permit.general, interlockJogForward := "Unit1.Em5.ControlNodes".cm.Interlock.magazine.permit.jogForward, interlockJogBackward := "Unit1.Em5.ControlNodes".cm.Interlock.magazine.permit.jogBackward, moduleAccessPoint := "Unit1.Em5.Config".moduleAccessPoint[2], axisNo :=, axis := "Unit1.Em5.Config".axis[2], configuration := "Unit1.Em5.Config".cmMagazineAxisZ, moduleInterface := "Unit1.Em5.HmiInterface".cmMagazineAxisZ, controlNode := "Unit1.Em5.ControlNodes".cmMagazineAxisZ, busy =>, actualPosition =>, actualSpeed =>)
   END_RUNG
   RUNG wire#powerrail
      Contact( #TRUE )
   END_RUNG wire#w1
   // the same network as SCL:
   #instCmMagazineAxisZ(enable := #TRUE,   // "LBC_Axis64Pos_TecPlcCn"
                        parentReferenceDesignator := "Unit1.Em5.Config".em.referenceDesignator.combined,
                        enableManualCmds := #statEnableManualCmds,
                        interlockGeneral := "Unit1.Em5.ControlNodes".cm.Interlock.magazine.permit.general,
                        interlockJogForward := "Unit1.Em5.ControlNodes".cm.Interlock.magazine.permit.jogForward,
                        interlockJogBackward := "Unit1.Em5.ControlNodes".cm.Interlock.magazine.permit.jogBackward,
                        moduleAccessPoint := "Unit1.Em5.Config".moduleAccessPoint[2],
                        axis := "Unit1.Em5.Config".axis[2],
                        configuration := "Unit1.Em5.Config".cmMagazineAxisZ,
                        moduleInterface := "Unit1.Em5.HmiInterface".cmMagazineAxisZ,
                        controlNode := "Unit1.Em5.ControlNodes".cmMagazineAxisZ);
END_REGION

REGION Network 55: Call CM Magazine Z Axis (LER_ServoTorqueCal)
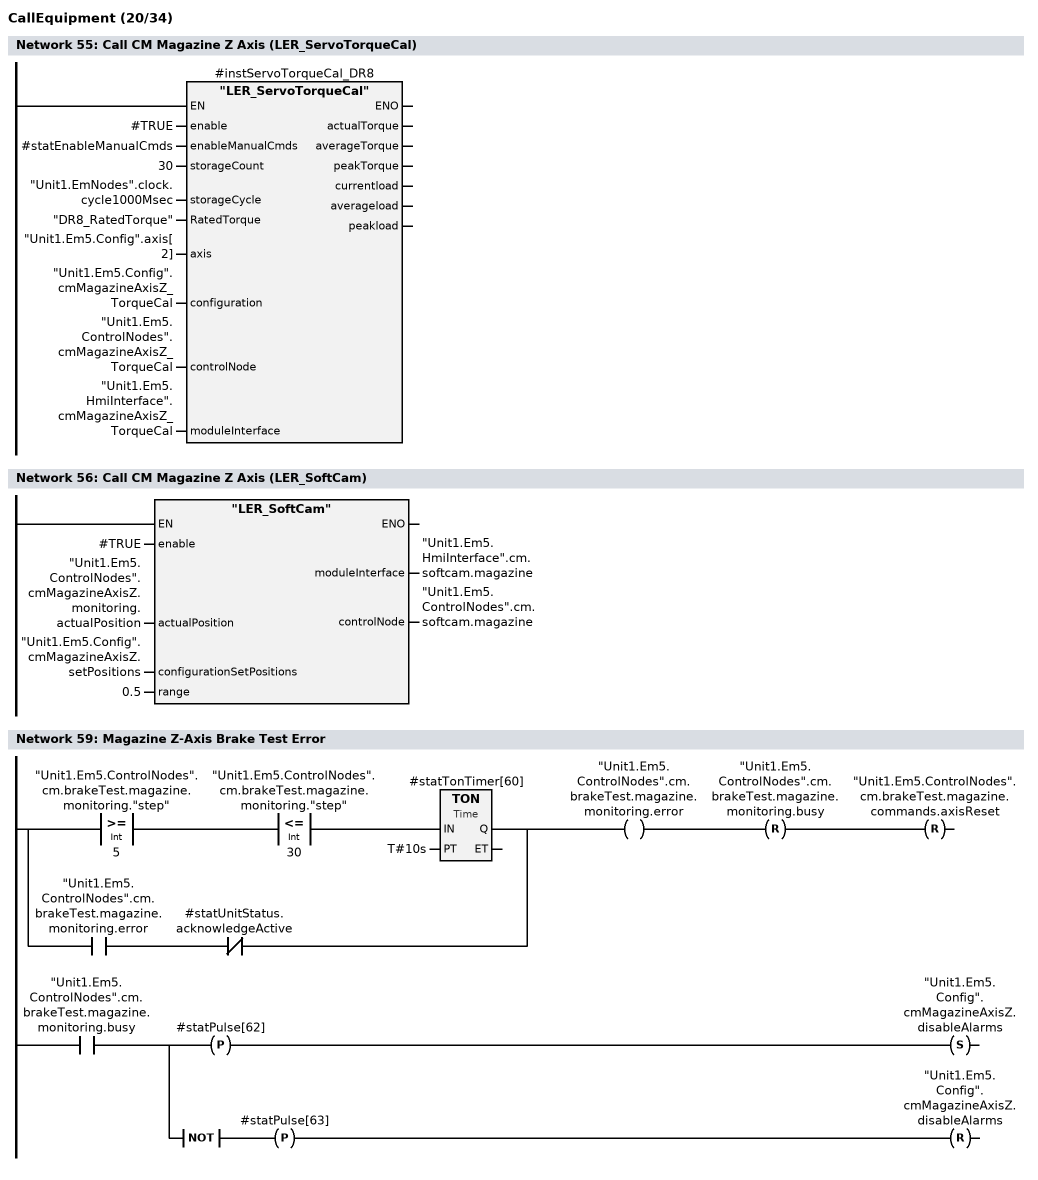
   RUNG wire#powerrail
      #instServoTorqueCal_DR8(enable := #TRUE, enableManualCmds := #statEnableManualCmds, storageCount := 30, storageCycle := "Unit1.EmNodes".clock.cycle1000Msec, RatedTorque := "DR8_RatedTorque", axis := "Unit1.Em5.Config".axis[2], configuration := "Unit1.Em5.Config".cmMagazineAxisZ_TorqueCal, controlNode := "Unit1.Em5.ControlNodes".cmMagazineAxisZ_TorqueCal, moduleInterface := "Unit1.Em5.HmiInterface".cmMagazineAxisZ_TorqueCal, actualTorque =>, averageTorque =>, peakTorque =>, currentload =>, averageload =>, peakload =>)
   END_RUNG
   // the same network as SCL:
   #instServoTorqueCal_DR8(enable := #TRUE,   // "LER_ServoTorqueCal"
                           enableManualCmds := #statEnableManualCmds,
                           storageCount := 30,
                           storageCycle := "Unit1.EmNodes".clock.cycle1000Msec,
                           RatedTorque := "DR8_RatedTorque",
                           axis := "Unit1.Em5.Config".axis[2],
                           configuration := "Unit1.Em5.Config".cmMagazineAxisZ_TorqueCal,
                           controlNode := "Unit1.Em5.ControlNodes".cmMagazineAxisZ_TorqueCal,
                           moduleInterface := "Unit1.Em5.HmiInterface".cmMagazineAxisZ_TorqueCal);
END_REGION

REGION Network 56: Call CM Magazine Z Axis (LER_SoftCam)
   RUNG wire#powerrail
      "LER_SoftCam"(enable := #TRUE, actualPosition := "Unit1.Em5.ControlNodes".cmMagazineAxisZ.monitoring.actualPosition, configurationSetPositions := "Unit1.Em5.Config".cmMagazineAxisZ.setPositions, range := 0.5, moduleInterface => "Unit1.Em5.HmiInterface".cm.softcam.magazine, controlNode => "Unit1.Em5.ControlNodes".cm.softcam.magazine)
   END_RUNG
   // the same network as SCL:
   "LER_SoftCam"(enable := #TRUE,
                 actualPosition := "Unit1.Em5.ControlNodes".cmMagazineAxisZ.monitoring.actualPosition,
                 configurationSetPositions := "Unit1.Em5.Config".cmMagazineAxisZ.setPositions,
                 range := 0.5,
                 moduleInterface => "Unit1.Em5.HmiInterface".cm.softcam.magazine,
                 controlNode => "Unit1.Em5.ControlNodes".cm.softcam.magazine);
END_REGION

REGION Network 58: ******************** Brake Test (Axis) ********************
END_REGION

